% RSLogix 500 project GILL ONION_11_12_2021_BAK142.RSS, saved by version 11.00.00.00 %
PROJECT "UNTITLED"    % processor: MicroLogix 1400 %

PROGRAM FILES
  LAD 2 "MAIN"  10 rungs
  LAD 3 "UNSTACKER"  32 rungs
  LAD 4 "BS"  36 rungs
  LAD 5 "STACKER"  32 rungs
  LAD 6 "WATER"  21 rungs
  LAD 7 "CONVEYORS"  1 rungs
  LAD 8 "ENCODER"  6 rungs  % Bin Scrubber HSC %
  LAD 9 "STARTUP"  6 rungs
  LAD 10 "FAULTS"  65 rungs  % Faults %
  LAD 11 "HSC"  2 rungs  % Bin Scrubber Cradle %

DATA FILES
  O0 OUTPUT  8 elements
  I1 INPUT  18 elements
  S2 STATUS  66 elements
  B3 BINARY  9 elements
  T4 TIMER  34 elements
  C5 COUNTER  1 elements
  R6 CONTROL  1 elements
  N7 INTEGER  21 elements
  F8 FLOAT  1 elements
  L9   3 elements

LADDER 2 "MAIN"
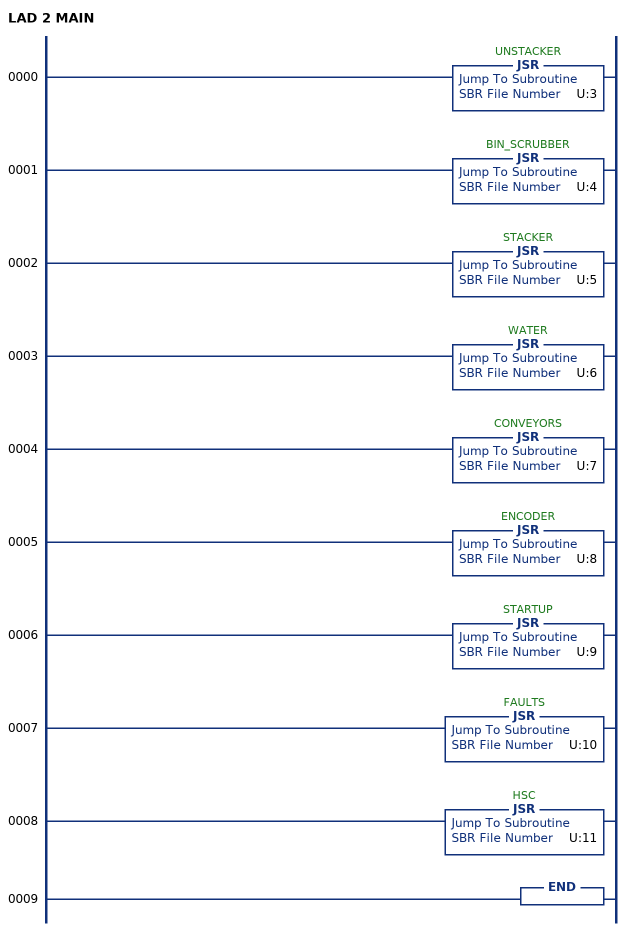
% Rung: 0 %
SOR JSR U:3 EOR
%   U:3  UNSTACKER %
% Rung: 1 %
SOR JSR U:4 EOR
%   U:4  BIN_SCRUBBER %
% Rung: 2 %
SOR JSR U:5 EOR
%   U:5  STACKER %
% Rung: 3 %
SOR JSR U:6 EOR
%   U:6  WATER %
% Rung: 4 %
SOR JSR U:7 EOR
%   U:7  CONVEYORS %
% Rung: 5 %
SOR JSR U:8 EOR
%   U:8  ENCODER %
% Rung: 6 %
SOR JSR U:9 EOR
%   U:9  STARTUP %
% Rung: 7 %
SOR JSR U:10 EOR
%   U:10  FAULTS %
% Rung: 8 %
SOR JSR U:11 EOR
%   U:11  HSC %
% Rung: 9 %
SOR END EOR

LADDER 3 "UNSTACKER"
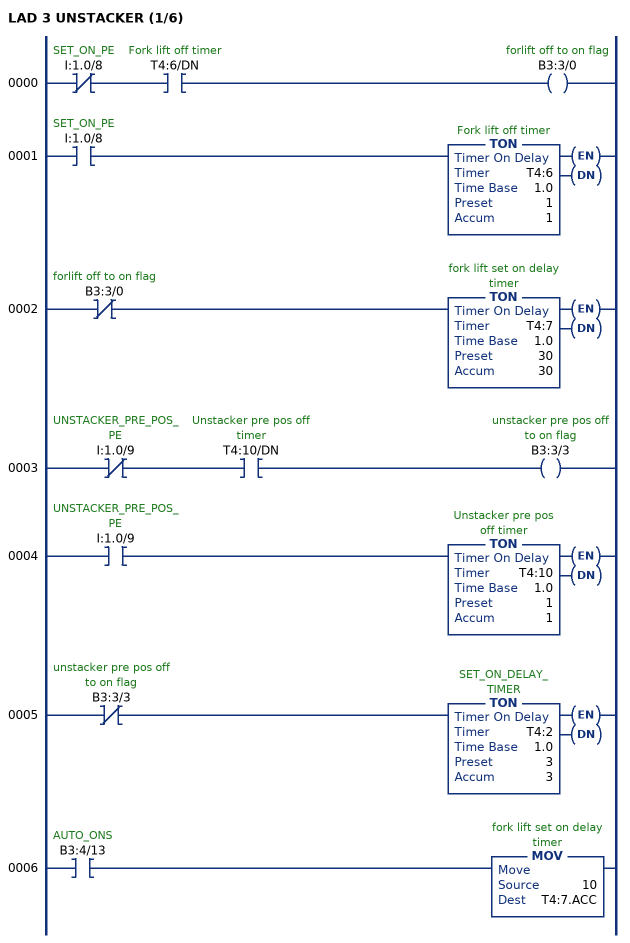
% Rung: 0 %
SOR XIO I:1.0/8 XIC T4:6/DN OTE B3:3/0 EOR
%   I:1.0/8  SET_ON_PE %
%   T4:6  "Fork lift off timer" %
%   B3:3/0  "forlift off to on flag" %
% Rung: 1 %
SOR XIC I:1.0/8 TON T4:6 1.0 1 1 EOR
%   I:1.0/8  SET_ON_PE %
%   T4:6  "Fork lift off timer" %
% Rung: 2 %
SOR XIO B3:3/0 TON T4:7 1.0 30 30 EOR
%   B3:3/0  "forlift off to on flag" %
%   T4:7  "fork lift set on delay timer" %
% Rung: 3 %
SOR XIO I:1.0/9 XIC T4:10/DN OTE B3:3/3 EOR
%   I:1.0/9  UNSTACKER_PRE_POS_PE %
%   T4:10  "Unstacker pre pos off timer" %
%   B3:3/3  "unstacker pre pos off to on flag" %
% Rung: 4 %
SOR XIC I:1.0/9 TON T4:10 1.0 1 1 EOR
%   I:1.0/9  UNSTACKER_PRE_POS_PE %
%   T4:10  "Unstacker pre pos off timer" %
% Rung: 5 %
SOR XIO B3:3/3 TON T4:2 1.0 3 3 EOR
%   B3:3/3  "unstacker pre pos off to on flag" %
%   T4:2  SET_ON_DELAY_TIMER %
% Rung: 6 %
SOR XIC B3:4/13 MOV 10 T4:7.ACC EOR
%   B3:4/13  AUTO_ONS %
%   T4:7  "fork lift set on delay timer" %

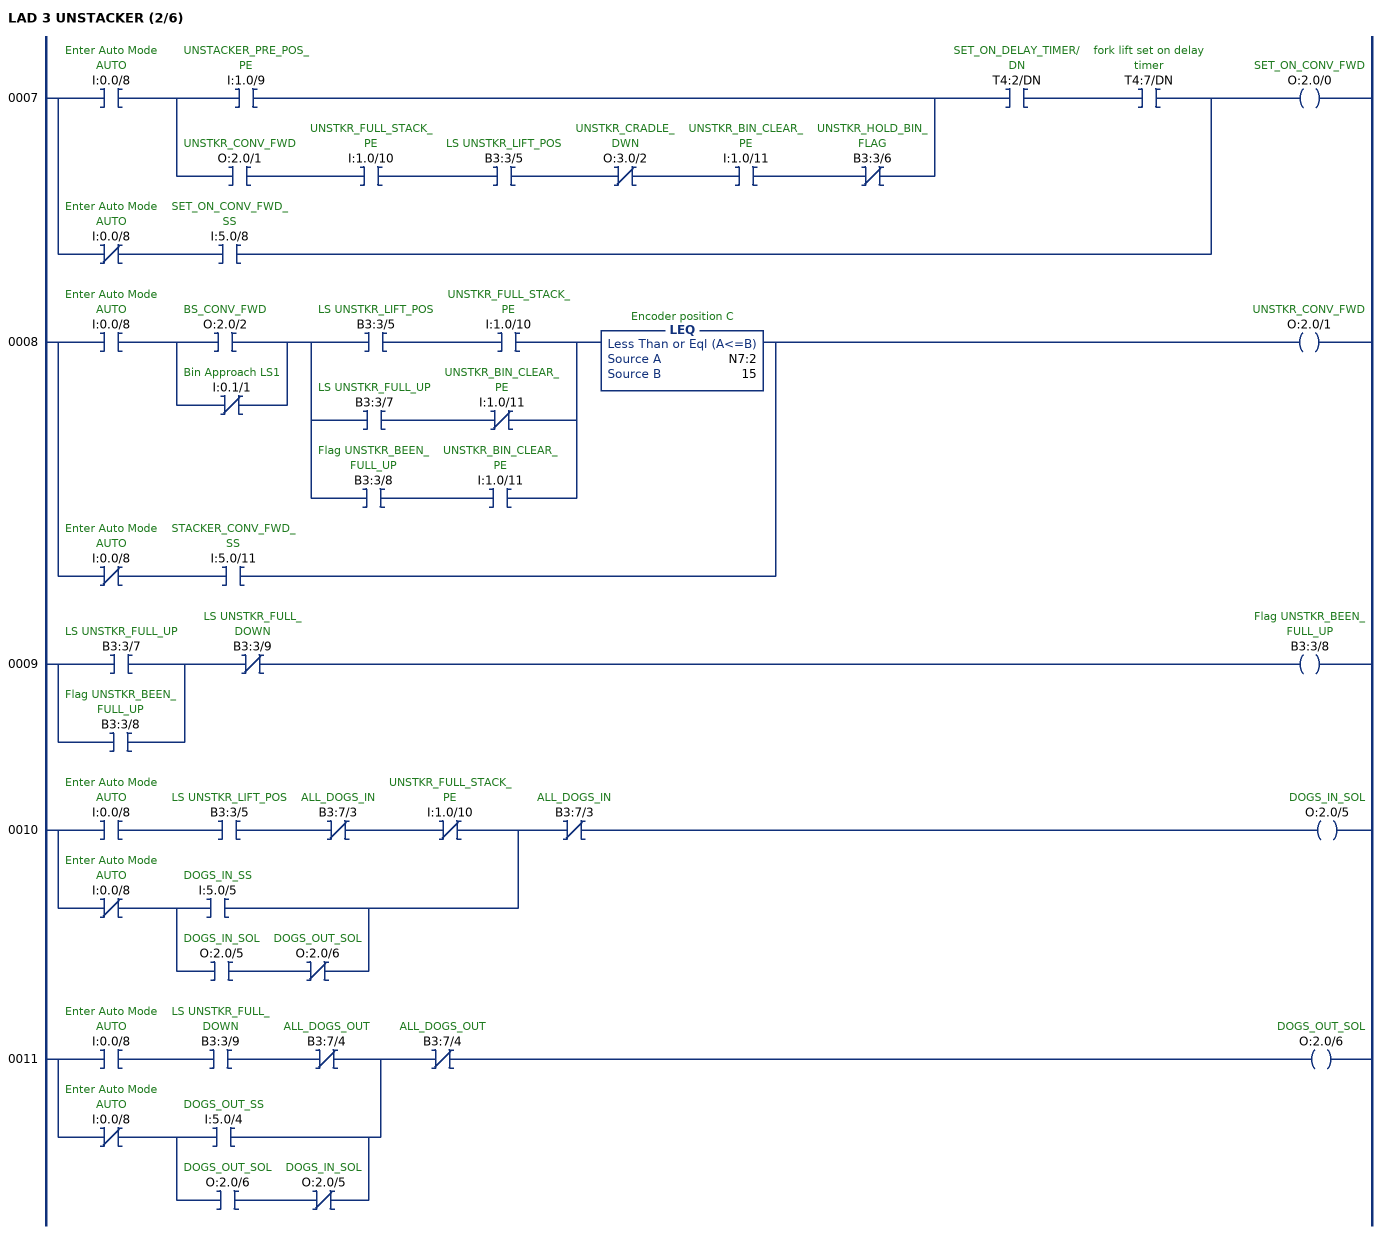
% Rung: 7 %
SOR BST XIC I:0.0/8 BST XIC I:1.0/9 NXB XIC O:2.0/1 XIC I:1.0/10 XIC B3:3/5 XIO O:3.0/2 XIC I:1.0/11 XIO B3:3/6 BND XIC T4:2/DN XIC T4:7/DN NXB XIO I:0.0/8 XIC I:5.0/8 BND OTE O:2.0/0 EOR
%   I:0.0/8  AUTO  "Enter Auto Mode" %
%   I:1.0/9  UNSTACKER_PRE_POS_PE %
%   O:2.0/1  UNSTKR_CONV_FWD %
%   I:1.0/10  UNSTKR_FULL_STACK_PE %
%   B3:3/5  UNSTKR_LIFT_POS  "LS" %
%   O:3.0/2  UNSTKR_CRADLE_DWN %
%   I:1.0/11  UNSTKR_BIN_CLEAR_PE %
%   B3:3/6  UNSTKR_HOLD_BIN_FLAG %
%   T4:2  SET_ON_DELAY_TIMER %
%   T4:7  "fork lift set on delay timer" %
%   I:5.0/8  SET_ON_CONV_FWD_SS %
%   O:2.0/0  SET_ON_CONV_FWD %
% Rung: 8 %
SOR BST XIC I:0.0/8 BST XIC O:2.0/2 NXB XIO I:0.1/1 BND BST XIC B3:3/5 XIC I:1.0/10 NXB BST XIC B3:3/7 XIO I:1.0/11 NXB XIC B3:3/8 XIC I:1.0/11 BND BND LEQ N7:2 15 NXB XIO I:0.0/8 XIC I:5.0/11 BND OTE O:2.0/1 EOR
%   I:0.0/8  AUTO  "Enter Auto Mode" %
%   O:2.0/2  BS_CONV_FWD %
%   I:0.1/1  LS1  "Bin Approach" %
%   B3:3/5  UNSTKR_LIFT_POS  "LS" %
%   I:1.0/10  UNSTKR_FULL_STACK_PE %
%   B3:3/7  UNSTKR_FULL_UP  "LS" %
%   I:1.0/11  UNSTKR_BIN_CLEAR_PE %
%   B3:3/8  UNSTKR_BEEN_FULL_UP  "Flag" %
%   N7:2  C  "Encoder position" %
%   I:5.0/11  STACKER_CONV_FWD_SS %
%   O:2.0/1  UNSTKR_CONV_FWD %
% Rung: 9 %
SOR BST XIC B3:3/7 NXB XIC B3:3/8 BND XIO B3:3/9 OTE B3:3/8 EOR
%   B3:3/7  UNSTKR_FULL_UP  "LS" %
%   B3:3/8  UNSTKR_BEEN_FULL_UP  "Flag" %
%   B3:3/9  UNSTKR_FULL_DOWN  "LS" %
% Rung: 10 %
SOR BST XIC I:0.0/8 XIC B3:3/5 XIO B3:7/3 XIO I:1.0/10 NXB XIO I:0.0/8 BST XIC I:5.0/5 NXB XIC O:2.0/5 XIO O:2.0/6 BND BND XIO B3:7/3 OTE O:2.0/5 EOR
%   I:0.0/8  AUTO  "Enter Auto Mode" %
%   B3:3/5  UNSTKR_LIFT_POS  "LS" %
%   B3:7/3  ALL_DOGS_IN %
%   I:1.0/10  UNSTKR_FULL_STACK_PE %
%   I:5.0/5  DOGS_IN_SS %
%   O:2.0/5  DOGS_IN_SOL %
%   O:2.0/6  DOGS_OUT_SOL %
% Rung: 11 %
SOR BST XIC I:0.0/8 XIC B3:3/9 XIO B3:7/4 NXB XIO I:0.0/8 BST XIC I:5.0/4 NXB XIC O:2.0/6 XIO O:2.0/5 BND BND XIO B3:7/4 OTE O:2.0/6 EOR
%   I:0.0/8  AUTO  "Enter Auto Mode" %
%   B3:3/9  UNSTKR_FULL_DOWN  "LS" %
%   B3:7/4  ALL_DOGS_OUT %
%   I:5.0/4  DOGS_OUT_SS %
%   O:2.0/6  DOGS_OUT_SOL %
%   O:2.0/5  DOGS_IN_SOL %

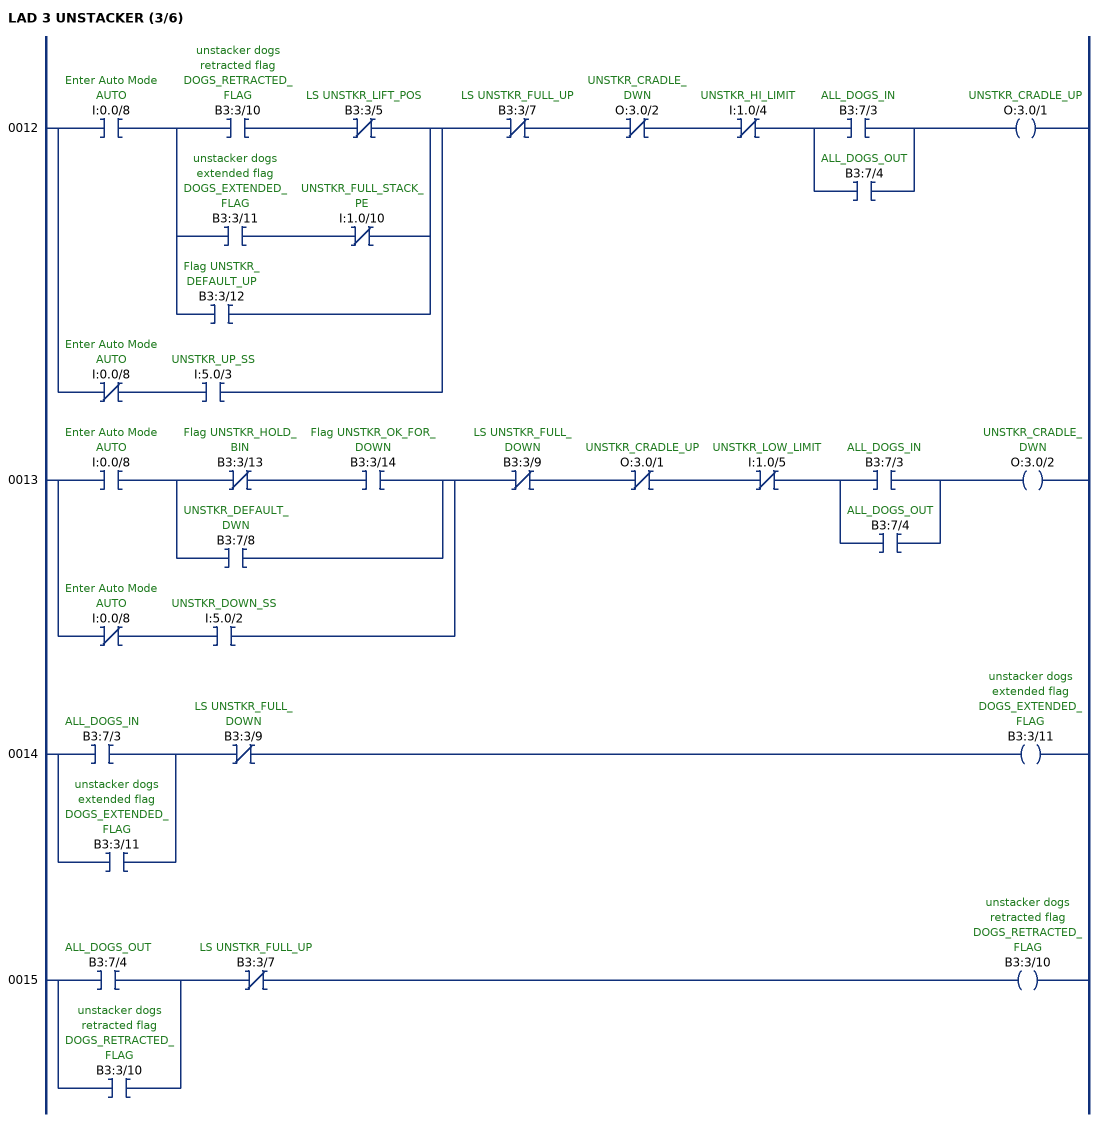
% Rung: 12 %
SOR BST XIC I:0.0/8 BST XIC B3:3/10 XIO B3:3/5 NXB BST XIC B3:3/11 XIO I:1.0/10 NXB XIC B3:3/12 BND BND NXB XIO I:0.0/8 XIC I:5.0/3 BND XIO B3:3/7 XIO O:3.0/2 XIO I:1.0/4 BST XIC B3:7/3 NXB XIC B3:7/4 BND OTE O:3.0/1 EOR
%   I:0.0/8  AUTO  "Enter Auto Mode" %
%   B3:3/10  DOGS_RETRACTED_FLAG  "unstacker dogs retracted flag" %
%   B3:3/5  UNSTKR_LIFT_POS  "LS" %
%   B3:3/11  DOGS_EXTENDED_FLAG  "unstacker dogs extended flag" %
%   I:1.0/10  UNSTKR_FULL_STACK_PE %
%   B3:3/12  UNSTKR_DEFAULT_UP  "Flag" %
%   I:5.0/3  UNSTKR_UP_SS %
%   B3:3/7  UNSTKR_FULL_UP  "LS" %
%   O:3.0/2  UNSTKR_CRADLE_DWN %
%   I:1.0/4  UNSTKR_HI_LIMIT %
%   B3:7/3  ALL_DOGS_IN %
%   B3:7/4  ALL_DOGS_OUT %
%   O:3.0/1  UNSTKR_CRADLE_UP %
% Rung: 13 %
SOR BST XIC I:0.0/8 BST XIO B3:3/13 XIC B3:3/14 NXB XIC B3:7/8 BND NXB XIO I:0.0/8 XIC I:5.0/2 BND XIO B3:3/9 XIO O:3.0/1 XIO I:1.0/5 BST XIC B3:7/3 NXB XIC B3:7/4 BND OTE O:3.0/2 EOR
%   I:0.0/8  AUTO  "Enter Auto Mode" %
%   B3:3/13  UNSTKR_HOLD_BIN  "Flag" %
%   B3:3/14  UNSTKR_OK_FOR_DOWN  "Flag" %
%   B3:7/8  UNSTKR_DEFAULT_DWN %
%   I:5.0/2  UNSTKR_DOWN_SS %
%   B3:3/9  UNSTKR_FULL_DOWN  "LS" %
%   O:3.0/1  UNSTKR_CRADLE_UP %
%   I:1.0/5  UNSTKR_LOW_LIMIT %
%   B3:7/3  ALL_DOGS_IN %
%   B3:7/4  ALL_DOGS_OUT %
%   O:3.0/2  UNSTKR_CRADLE_DWN %
% Rung: 14 %
SOR BST XIC B3:7/3 NXB XIC B3:3/11 BND XIO B3:3/9 OTE B3:3/11 EOR
%   B3:7/3  ALL_DOGS_IN %
%   B3:3/11  DOGS_EXTENDED_FLAG  "unstacker dogs extended flag" %
%   B3:3/9  UNSTKR_FULL_DOWN  "LS" %
% Rung: 15 %
SOR BST XIC B3:7/4 NXB XIC B3:3/10 BND XIO B3:3/7 OTE B3:3/10 EOR
%   B3:7/4  ALL_DOGS_OUT %
%   B3:3/10  DOGS_RETRACTED_FLAG  "unstacker dogs retracted flag" %
%   B3:3/7  UNSTKR_FULL_UP  "LS" %

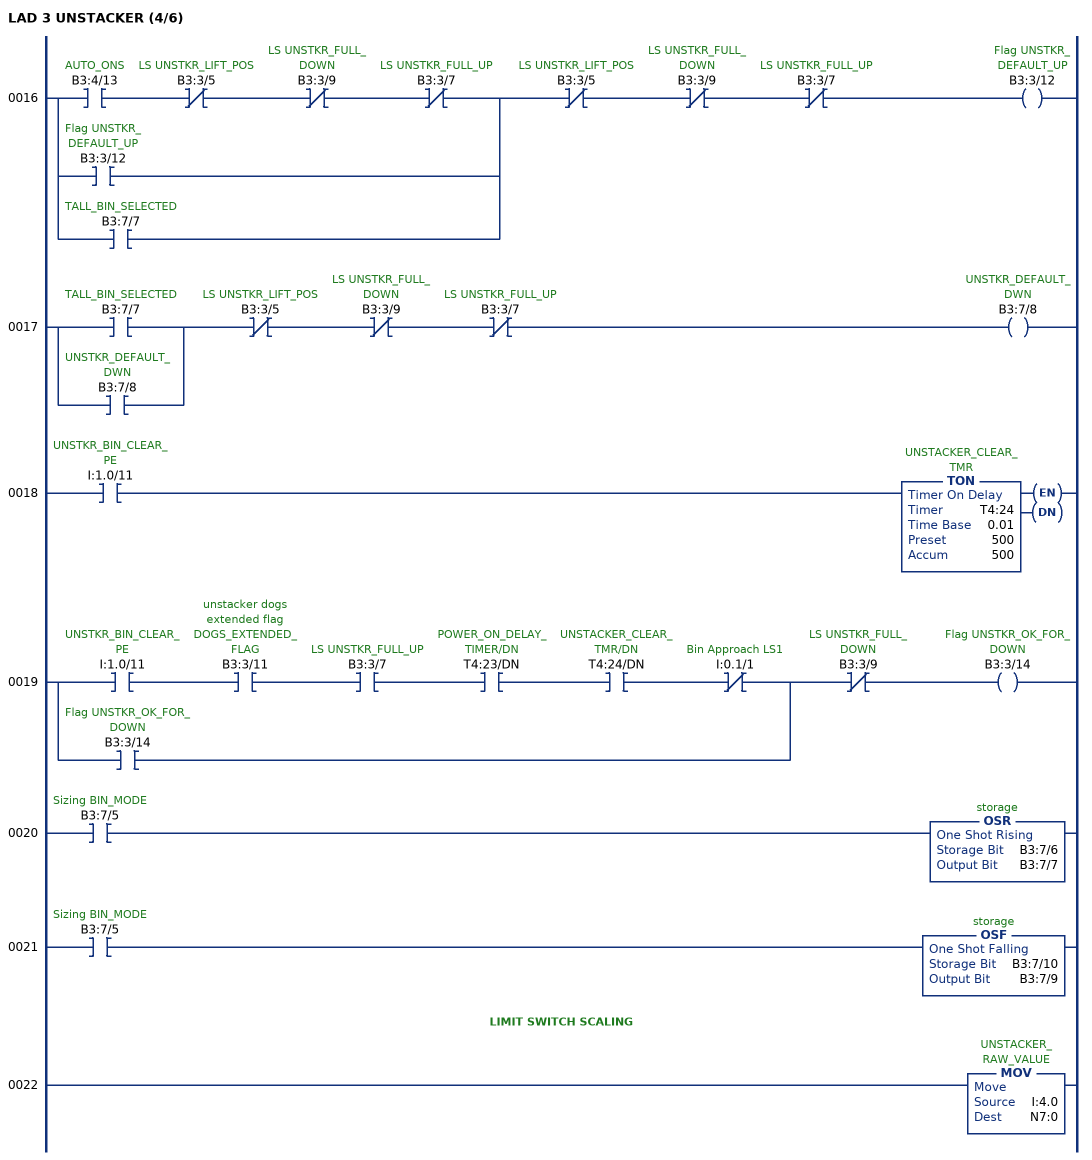
% Rung: 16 %
SOR BST XIC B3:4/13 XIO B3:3/5 XIO B3:3/9 XIO B3:3/7 NXB BST XIC B3:3/12 NXB XIC B3:7/7 BND BND XIO B3:3/5 XIO B3:3/9 XIO B3:3/7 OTE B3:3/12 EOR
%   B3:4/13  AUTO_ONS %
%   B3:3/5  UNSTKR_LIFT_POS  "LS" %
%   B3:3/9  UNSTKR_FULL_DOWN  "LS" %
%   B3:3/7  UNSTKR_FULL_UP  "LS" %
%   B3:3/12  UNSTKR_DEFAULT_UP  "Flag" %
%   B3:7/7  TALL_BIN_SELECTED %
% Rung: 17 %
SOR BST XIC B3:7/7 NXB XIC B3:7/8 BND XIO B3:3/5 XIO B3:3/9 XIO B3:3/7 OTE B3:7/8 EOR
%   B3:7/7  TALL_BIN_SELECTED %
%   B3:7/8  UNSTKR_DEFAULT_DWN %
%   B3:3/5  UNSTKR_LIFT_POS  "LS" %
%   B3:3/9  UNSTKR_FULL_DOWN  "LS" %
%   B3:3/7  UNSTKR_FULL_UP  "LS" %
% Rung: 18 %
SOR XIC I:1.0/11 TON T4:24 0.01 500 500 EOR
%   I:1.0/11  UNSTKR_BIN_CLEAR_PE %
%   T4:24  UNSTACKER_CLEAR_TMR %
% Rung: 19 %
SOR BST XIC I:1.0/11 XIC B3:3/11 XIC B3:3/7 XIC T4:23/DN XIC T4:24/DN XIO I:0.1/1 NXB XIC B3:3/14 BND XIO B3:3/9 OTE B3:3/14 EOR
%   I:1.0/11  UNSTKR_BIN_CLEAR_PE %
%   B3:3/11  DOGS_EXTENDED_FLAG  "unstacker dogs extended flag" %
%   B3:3/7  UNSTKR_FULL_UP  "LS" %
%   T4:23  POWER_ON_DELAY_TIMER %
%   T4:24  UNSTACKER_CLEAR_TMR %
%   I:0.1/1  LS1  "Bin Approach" %
%   B3:3/14  UNSTKR_OK_FOR_DOWN  "Flag" %
%   B3:3/9  UNSTKR_FULL_DOWN  "LS" %
% Rung: 20 %
SOR XIC B3:7/5 OSR B3:7/6 B3:7/7 EOR
%   B3:7/5  BIN_MODE  "Sizing" %
%   B3:7/6  "storage" %
%   B3:7/7  TALL_BIN_SELECTED %
% Rung: 21 %
SOR XIC B3:7/5 OSF B3:7/10 B3:7/9 EOR
%   B3:7/5  BIN_MODE  "Sizing" %
%   B3:7/10  "storage" %
%   B3:7/9  SMALL_BIN_SELECTED %
% Rung: 22 %
% TITLE: LIMIT SWITCH SCALING %
SOR MOV I:4.0 N7:0 EOR
%   I:4.0  UNSTACKER_RAW  "Draw String Encoder" %
%   N7:0  UNSTACKER_RAW_VALUE %

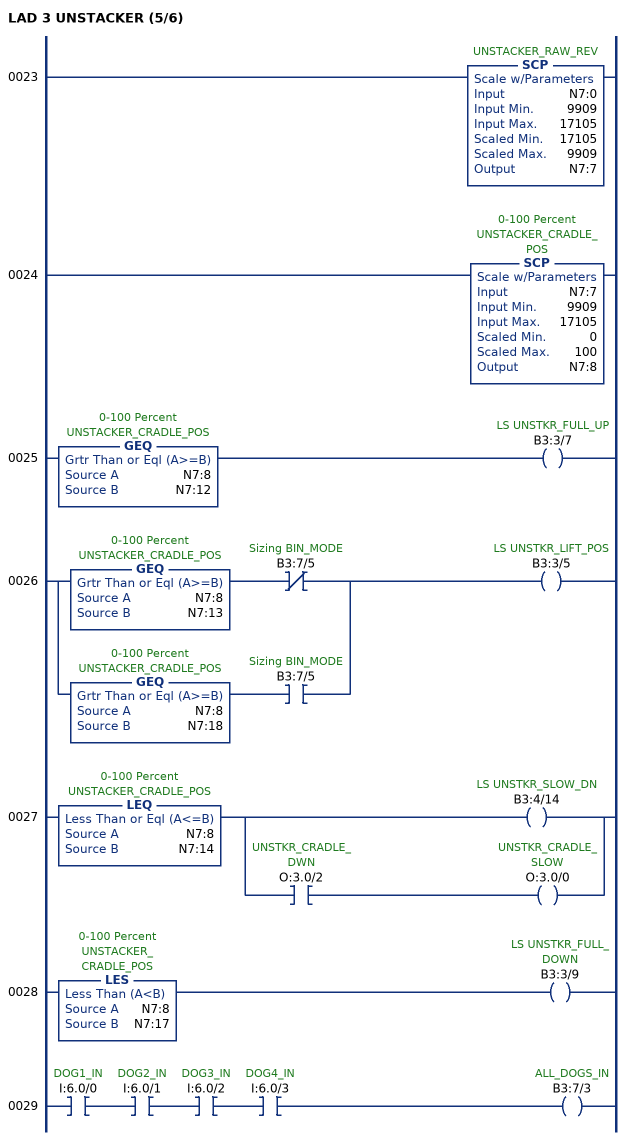
% Rung: 23 %
SOR SCP N7:0 9909 17105 17105 9909 N7:7 EOR
%   N7:0  UNSTACKER_RAW_VALUE %
%   N7:7  UNSTACKER_RAW_REV %
% Rung: 24 %
SOR SCP N7:7 9909 17105 0 100 N7:8 EOR
%   N7:7  UNSTACKER_RAW_REV %
%   N7:8  UNSTACKER_CRADLE_POS  "0-100 Percent" %
% Rung: 25 %
SOR GEQ N7:8 N7:12 OTE B3:3/7 EOR
%   N7:8  UNSTACKER_CRADLE_POS  "0-100 Percent" %
%   N7:12  UNSTKR_FULL_UP_SP  "Unstacker" %
%   B3:3/7  UNSTKR_FULL_UP  "LS" %
% Rung: 26 %
SOR BST GEQ N7:8 N7:13 XIO B3:7/5 NXB GEQ N7:8 N7:18 XIC B3:7/5 BND OTE B3:3/5 EOR
%   N7:8  UNSTACKER_CRADLE_POS  "0-100 Percent" %
%   N7:13  UNSTACKER_LIFT_SP  "Unstacker Lift Pos" %
%   B3:7/5  BIN_MODE  "Sizing" %
%   N7:18  TALL_BIN_SP %
%   B3:3/5  UNSTKR_LIFT_POS  "LS" %
% Rung: 27 %
SOR LEQ N7:8 N7:14 BST OTE B3:4/14 NXB XIC O:3.0/2 OTE O:3.0/0 BND EOR
%   N7:8  UNSTACKER_CRADLE_POS  "0-100 Percent" %
%   N7:14  UNSTKR_FULL_DOWN_SP  "Unstacker Full Down" %
%   B3:4/14  UNSTKR_SLOW_DN  "LS" %
%   O:3.0/2  UNSTKR_CRADLE_DWN %
%   O:3.0/0  UNSTKR_CRADLE_SLOW %
% Rung: 28 %
SOR LES N7:8 N7:17 OTE B3:3/9 EOR
%   N7:8  UNSTACKER_CRADLE_POS  "0-100 Percent" %
%   N7:17  "Unstacker" %
%   B3:3/9  UNSTKR_FULL_DOWN  "LS" %
% Rung: 29 %
SOR XIC I:6.0/0 XIC I:6.0/1 XIC I:6.0/2 XIC I:6.0/3 OTE B3:7/3 EOR
%   I:6.0/0  DOG1_IN %
%   I:6.0/1  DOG2_IN %
%   I:6.0/2  DOG3_IN %
%   I:6.0/3  DOG4_IN %
%   B3:7/3  ALL_DOGS_IN %

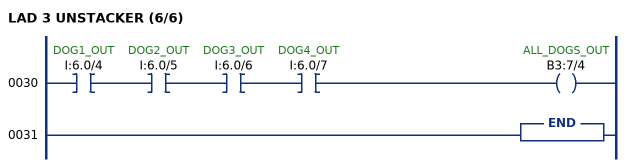
% Rung: 30 %
SOR XIC I:6.0/4 XIC I:6.0/5 XIC I:6.0/6 XIC I:6.0/7 OTE B3:7/4 EOR
%   I:6.0/4  DOG1_OUT %
%   I:6.0/5  DOG2_OUT %
%   I:6.0/6  DOG3_OUT %
%   I:6.0/7  DOG4_OUT %
%   B3:7/4  ALL_DOGS_OUT %
% Rung: 31 %
SOR END EOR

LADDER 4 "BS"
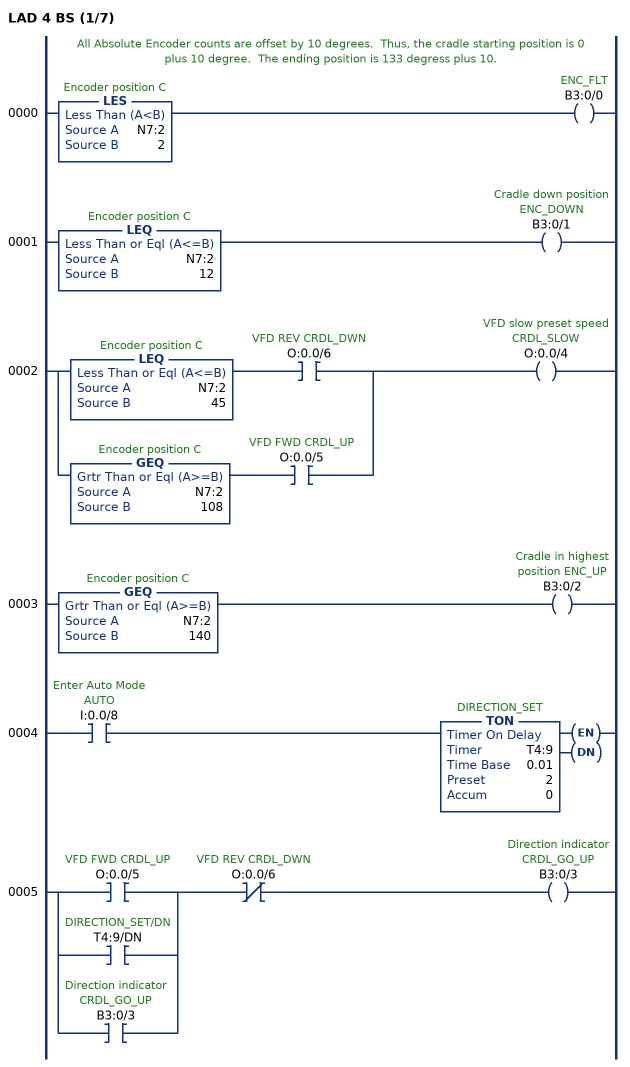
% Rung: 0 %
% All Absolute Encoder counts are offset by 10 degrees.  Thus, the cradle starting position is 0 plus 10 degree.  The ending position is 133 degress plus 10. %
SOR LES N7:2 2 OTE B3:0/0 EOR
%   N7:2  C  "Encoder position" %
%   B3:0/0  ENC_FLT %
% Rung: 1 %
SOR LEQ N7:2 12 OTE B3:0/1 EOR
%   N7:2  C  "Encoder position" %
%   B3:0/1  ENC_DOWN  "Cradle down position" %
% Rung: 2 %
SOR BST LEQ N7:2 45 XIC O:0.0/6 NXB GEQ N7:2 108 XIC O:0.0/5 BND OTE O:0.0/4 EOR
%   N7:2  C  "Encoder position" %
%   O:0.0/6  CRDL_DWN  "VFD REV" %
%   O:0.0/5  CRDL_UP  "VFD FWD" %
%   O:0.0/4  CRDL_SLOW  "VFD slow preset speed" %
% Rung: 3 %
SOR GEQ N7:2 140 OTE B3:0/2 EOR
%   N7:2  C  "Encoder position" %
%   B3:0/2  ENC_UP  "Cradle in highest position" %
% Rung: 4 %
SOR XIC I:0.0/8 TON T4:9 0.01 2 0 EOR
%   I:0.0/8  AUTO  "Enter Auto Mode" %
%   T4:9  DIRECTION_SET %
% Rung: 5 %
SOR BST XIC O:0.0/5 NXB XIC T4:9/DN NXB XIC B3:0/3 BND XIO O:0.0/6 OTE B3:0/3 EOR
%   O:0.0/5  CRDL_UP  "VFD FWD" %
%   T4:9  DIRECTION_SET %
%   B3:0/3  CRDL_GO_UP  "Direction indicator" %
%   O:0.0/6  CRDL_DWN  "VFD REV" %

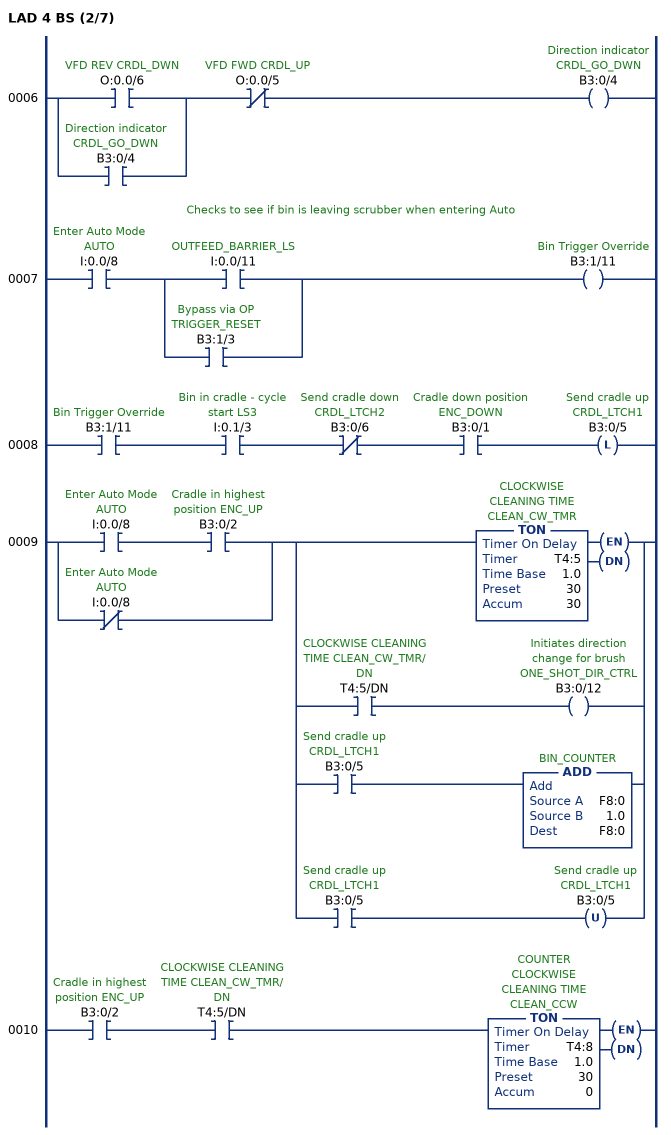
% Rung: 6 %
SOR BST XIC O:0.0/6 NXB XIC B3:0/4 BND XIO O:0.0/5 OTE B3:0/4 EOR
%   O:0.0/6  CRDL_DWN  "VFD REV" %
%   B3:0/4  CRDL_GO_DWN  "Direction indicator" %
%   O:0.0/5  CRDL_UP  "VFD FWD" %
% Rung: 7 %
% Checks to see if bin is leaving scrubber when entering Auto %
SOR XIC I:0.0/8 BST XIC I:0.0/11 NXB XIC B3:1/3 BND OTE B3:1/11 EOR
%   I:0.0/8  AUTO  "Enter Auto Mode" %
%   I:0.0/11  OUTFEED_BARRIER_LS %
%   B3:1/3  TRIGGER_RESET  "Bypass via OP" %
%   B3:1/11  "Bin Trigger Override" %
% Rung: 8 %
SOR XIC B3:1/11 XIC I:0.1/3 XIO B3:0/6 XIC B3:0/1 OTL B3:0/5 EOR
%   B3:1/11  "Bin Trigger Override" %
%   I:0.1/3  LS3  "Bin in cradle - cycle start" %
%   B3:0/6  CRDL_LTCH2  "Send cradle down" %
%   B3:0/1  ENC_DOWN  "Cradle down position" %
%   B3:0/5  CRDL_LTCH1  "Send cradle up" %
% Rung: 9 %
SOR BST XIC I:0.0/8 XIC B3:0/2 NXB XIO I:0.0/8 BND BST TON T4:5 1.0 30 30 NXB XIC T4:5/DN OTE B3:0/12 NXB BST XIC B3:0/5 ADD F8:0 1.0 F8:0 NXB XIC B3:0/5 OTU B3:0/5 BND BND EOR
%   I:0.0/8  AUTO  "Enter Auto Mode" %
%   B3:0/2  ENC_UP  "Cradle in highest position" %
%   T4:5  CLEAN_CW_TMR  "CLOCKWISE CLEANING TIME" %
%   B3:0/12  ONE_SHOT_DIR_CTRL  "Initiates direction change for brush" %
%   B3:0/5  CRDL_LTCH1  "Send cradle up" %
%   F8:0  BIN_COUNTER %
% Rung: 10 %
SOR XIC B3:0/2 XIC T4:5/DN TON T4:8 1.0 30 0 EOR
%   B3:0/2  ENC_UP  "Cradle in highest position" %
%   T4:5  CLEAN_CW_TMR  "CLOCKWISE CLEANING TIME" %
%   T4:8  CLEAN_CCW  "COUNTER CLOCKWISE CLEANING TIME" %

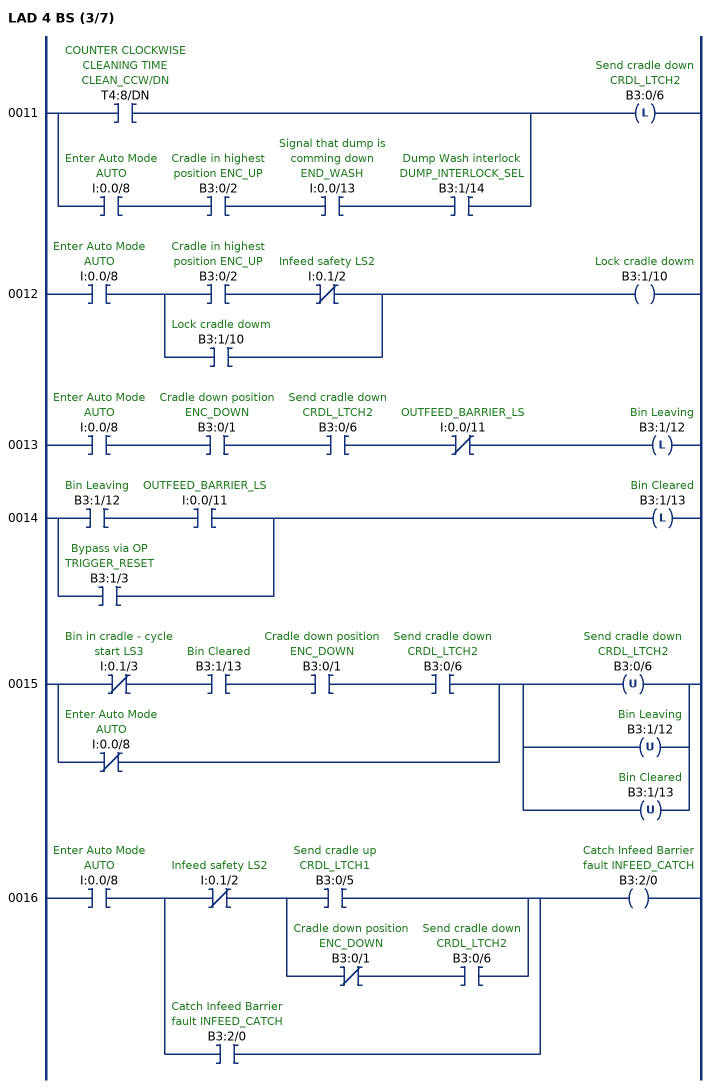
% Rung: 11 %
SOR BST XIC T4:8/DN NXB XIC I:0.0/8 XIC B3:0/2 XIC I:0.0/13 XIC B3:1/14 BND OTL B3:0/6 EOR
%   T4:8  CLEAN_CCW  "COUNTER CLOCKWISE CLEANING TIME" %
%   I:0.0/8  AUTO  "Enter Auto Mode" %
%   B3:0/2  ENC_UP  "Cradle in highest position" %
%   I:0.0/13  END_WASH  "Signal that dump is comming down" %
%   B3:1/14  DUMP_INTERLOCK_SEL  "Dump Wash interlock" %
%   B3:0/6  CRDL_LTCH2  "Send cradle down" %
% Rung: 12 %
SOR XIC I:0.0/8 BST XIC B3:0/2 XIO I:0.1/2 NXB XIC B3:1/10 BND OTE B3:1/10 EOR
%   I:0.0/8  AUTO  "Enter Auto Mode" %
%   B3:0/2  ENC_UP  "Cradle in highest position" %
%   I:0.1/2  LS2  "Infeed safety" %
%   B3:1/10  "Lock cradle dowm" %
% Rung: 13 %
SOR XIC I:0.0/8 XIC B3:0/1 XIC B3:0/6 XIO I:0.0/11 OTL B3:1/12 EOR
%   I:0.0/8  AUTO  "Enter Auto Mode" %
%   B3:0/1  ENC_DOWN  "Cradle down position" %
%   B3:0/6  CRDL_LTCH2  "Send cradle down" %
%   I:0.0/11  OUTFEED_BARRIER_LS %
%   B3:1/12  "Bin Leaving" %
% Rung: 14 %
SOR BST XIC B3:1/12 XIC I:0.0/11 NXB XIC B3:1/3 BND OTL B3:1/13 EOR
%   B3:1/12  "Bin Leaving" %
%   I:0.0/11  OUTFEED_BARRIER_LS %
%   B3:1/3  TRIGGER_RESET  "Bypass via OP" %
%   B3:1/13  "Bin Cleared" %
% Rung: 15 %
SOR BST XIO I:0.1/3 XIC B3:1/13 XIC B3:0/1 XIC B3:0/6 NXB XIO I:0.0/8 BND BST OTU B3:0/6 NXB BST OTU B3:1/12 NXB OTU B3:1/13 BND BND EOR
%   I:0.1/3  LS3  "Bin in cradle - cycle start" %
%   B3:1/13  "Bin Cleared" %
%   B3:0/1  ENC_DOWN  "Cradle down position" %
%   B3:0/6  CRDL_LTCH2  "Send cradle down" %
%   I:0.0/8  AUTO  "Enter Auto Mode" %
%   B3:1/12  "Bin Leaving" %
% Rung: 16 %
SOR XIC I:0.0/8 BST XIO I:0.1/2 BST XIC B3:0/5 NXB XIO B3:0/1 XIC B3:0/6 BND NXB XIC B3:2/0 BND OTE B3:2/0 EOR
%   I:0.0/8  AUTO  "Enter Auto Mode" %
%   I:0.1/2  LS2  "Infeed safety" %
%   B3:0/5  CRDL_LTCH1  "Send cradle up" %
%   B3:0/1  ENC_DOWN  "Cradle down position" %
%   B3:0/6  CRDL_LTCH2  "Send cradle down" %
%   B3:2/0  INFEED_CATCH  "Catch Infeed Barrier fault" %

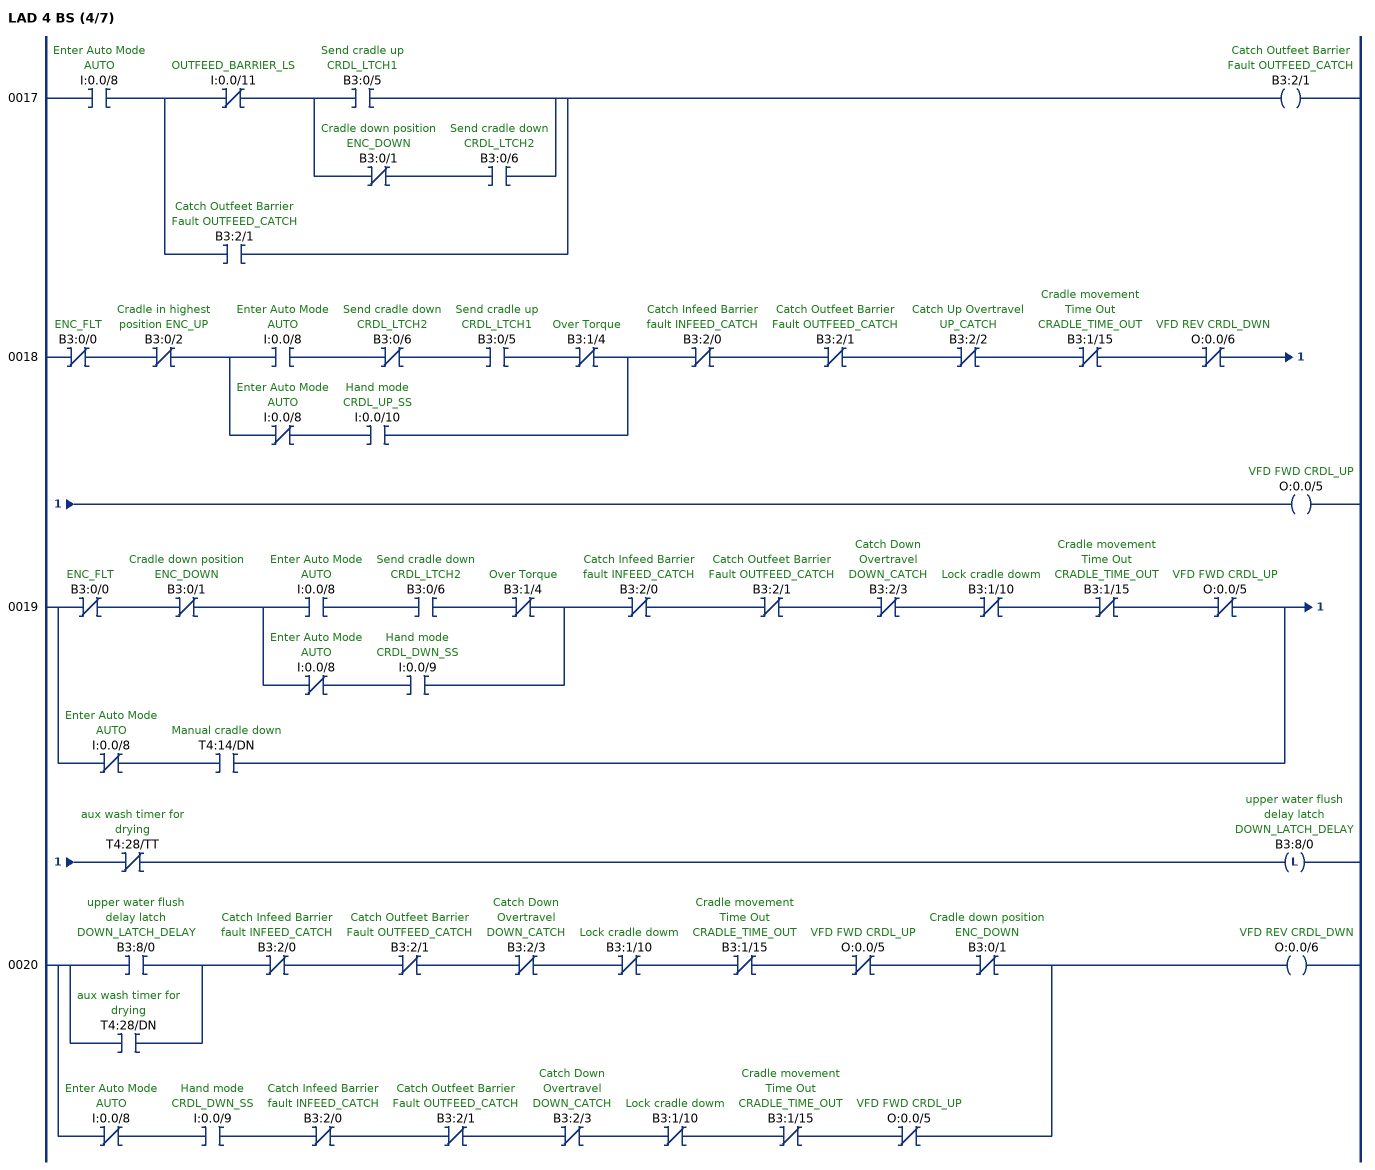
% Rung: 17 %
SOR XIC I:0.0/8 BST XIO I:0.0/11 BST XIC B3:0/5 NXB XIO B3:0/1 XIC B3:0/6 BND NXB XIC B3:2/1 BND OTE B3:2/1 EOR
%   I:0.0/8  AUTO  "Enter Auto Mode" %
%   I:0.0/11  OUTFEED_BARRIER_LS %
%   B3:0/5  CRDL_LTCH1  "Send cradle up" %
%   B3:0/1  ENC_DOWN  "Cradle down position" %
%   B3:0/6  CRDL_LTCH2  "Send cradle down" %
%   B3:2/1  OUTFEED_CATCH  "Catch Outfeet Barrier Fault" %
% Rung: 18 %
SOR XIO B3:0/0 XIO B3:0/2 BST XIC I:0.0/8 XIO B3:0/6 XIC B3:0/5 XIO B3:1/4 NXB XIO I:0.0/8 XIC I:0.0/10 BND XIO B3:2/0 XIO B3:2/1 XIO B3:2/2 XIO B3:1/15 XIO O:0.0/6 OTE O:0.0/5 EOR
%   B3:0/0  ENC_FLT %
%   B3:0/2  ENC_UP  "Cradle in highest position" %
%   I:0.0/8  AUTO  "Enter Auto Mode" %
%   B3:0/6  CRDL_LTCH2  "Send cradle down" %
%   B3:0/5  CRDL_LTCH1  "Send cradle up" %
%   B3:1/4  "Over Torque" %
%   I:0.0/10  CRDL_UP_SS  "Hand mode" %
%   B3:2/0  INFEED_CATCH  "Catch Infeed Barrier fault" %
%   B3:2/1  OUTFEED_CATCH  "Catch Outfeet Barrier Fault" %
%   B3:2/2  UP_CATCH  "Catch Up Overtravel" %
%   B3:1/15  CRADLE_TIME_OUT  "Cradle movement Time Out" %
%   O:0.0/6  CRDL_DWN  "VFD REV" %
%   O:0.0/5  CRDL_UP  "VFD FWD" %
% Rung: 19 %
SOR BST XIO B3:0/0 XIO B3:0/1 BST XIC I:0.0/8 XIC B3:0/6 XIO B3:1/4 NXB XIO I:0.0/8 XIC I:0.0/9 BND XIO B3:2/0 XIO B3:2/1 XIO B3:2/3 XIO B3:1/10 XIO B3:1/15 XIO O:0.0/5 NXB XIO I:0.0/8 XIC T4:14/DN BND XIO T4:28/TT OTL B3:8/0 EOR
%   B3:0/0  ENC_FLT %
%   B3:0/1  ENC_DOWN  "Cradle down position" %
%   I:0.0/8  AUTO  "Enter Auto Mode" %
%   B3:0/6  CRDL_LTCH2  "Send cradle down" %
%   B3:1/4  "Over Torque" %
%   I:0.0/9  CRDL_DWN_SS  "Hand mode" %
%   B3:2/0  INFEED_CATCH  "Catch Infeed Barrier fault" %
%   B3:2/1  OUTFEED_CATCH  "Catch Outfeet Barrier Fault" %
%   B3:2/3  DOWN_CATCH  "Catch Down Overtravel" %
%   B3:1/10  "Lock cradle dowm" %
%   B3:1/15  CRADLE_TIME_OUT  "Cradle movement Time Out" %
%   O:0.0/5  CRDL_UP  "VFD FWD" %
%   T4:14  "Manual cradle down" %
%   T4:28  "aux wash timer for drying" %
%   B3:8/0  DOWN_LATCH_DELAY  "upper water flush delay latch" %
% Rung: 20 %
SOR BST BST XIC B3:8/0 NXB XIC T4:28/DN BND XIO B3:2/0 XIO B3:2/1 XIO B3:2/3 XIO B3:1/10 XIO B3:1/15 XIO O:0.0/5 XIO B3:0/1 NXB XIO I:0.0/8 XIC I:0.0/9 XIO B3:2/0 XIO B3:2/1 XIO B3:2/3 XIO B3:1/10 XIO B3:1/15 XIO O:0.0/5 BND OTE O:0.0/6 EOR
%   B3:8/0  DOWN_LATCH_DELAY  "upper water flush delay latch" %
%   T4:28  "aux wash timer for drying" %
%   B3:2/0  INFEED_CATCH  "Catch Infeed Barrier fault" %
%   B3:2/1  OUTFEED_CATCH  "Catch Outfeet Barrier Fault" %
%   B3:2/3  DOWN_CATCH  "Catch Down Overtravel" %
%   B3:1/10  "Lock cradle dowm" %
%   B3:1/15  CRADLE_TIME_OUT  "Cradle movement Time Out" %
%   O:0.0/5  CRDL_UP  "VFD FWD" %
%   B3:0/1  ENC_DOWN  "Cradle down position" %
%   I:0.0/8  AUTO  "Enter Auto Mode" %
%   I:0.0/9  CRDL_DWN_SS  "Hand mode" %
%   O:0.0/6  CRDL_DWN  "VFD REV" %

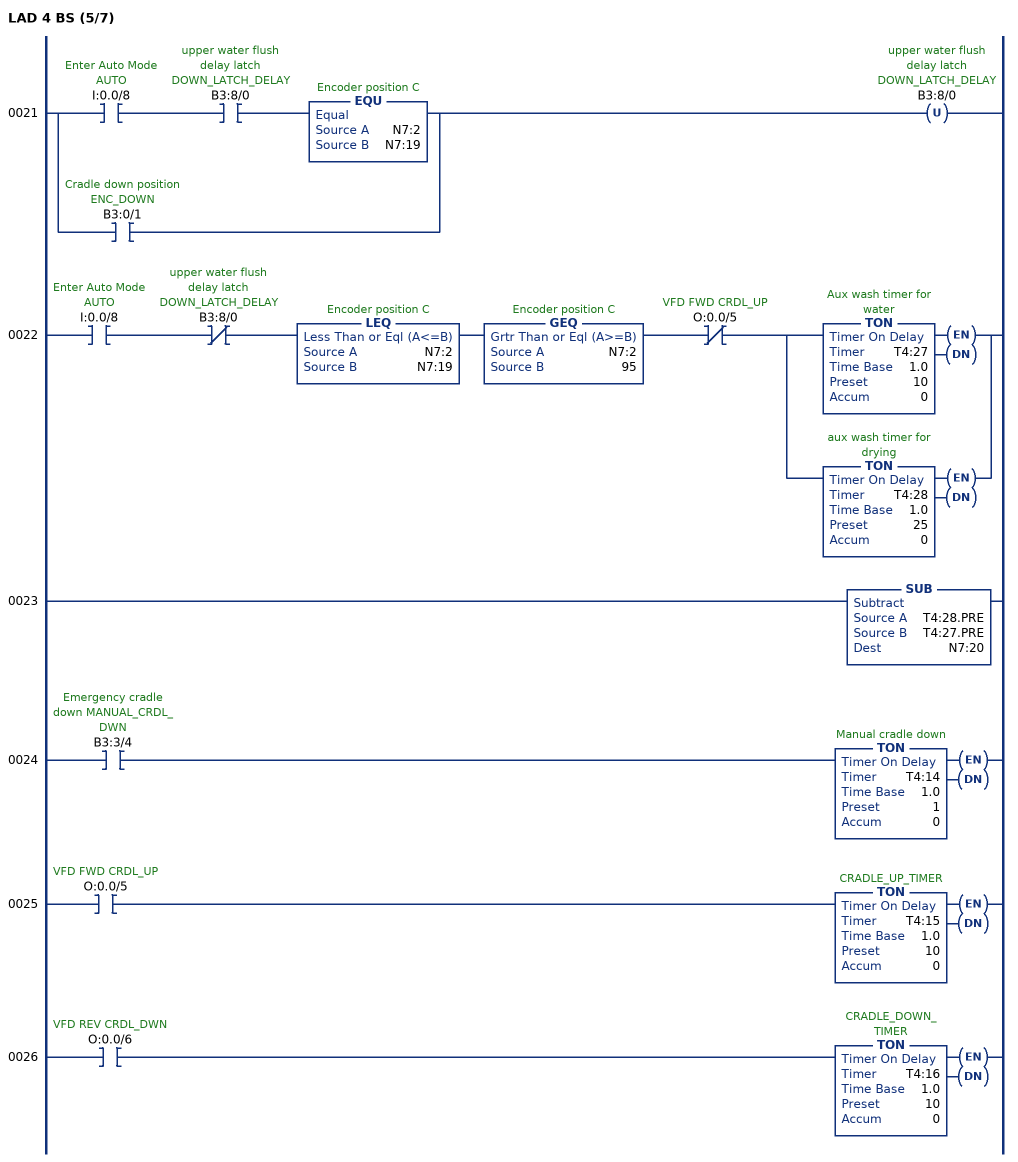
% Rung: 21 %
SOR BST XIC I:0.0/8 XIC B3:8/0 EQU N7:2 N7:19 NXB XIC B3:0/1 BND OTU B3:8/0 EOR
%   I:0.0/8  AUTO  "Enter Auto Mode" %
%   B3:8/0  DOWN_LATCH_DELAY  "upper water flush delay latch" %
%   N7:2  C  "Encoder position" %
%   N7:19  UPPER_WASH_SET_POINT  "HMI input for aux upper wash" %
%   B3:0/1  ENC_DOWN  "Cradle down position" %
% Rung: 22 %
SOR XIC I:0.0/8 XIO B3:8/0 LEQ N7:2 N7:19 GEQ N7:2 95 XIO O:0.0/5 BST TON T4:27 1.0 10 0 NXB TON T4:28 1.0 25 0 BND EOR
%   I:0.0/8  AUTO  "Enter Auto Mode" %
%   B3:8/0  DOWN_LATCH_DELAY  "upper water flush delay latch" %
%   N7:2  C  "Encoder position" %
%   N7:19  UPPER_WASH_SET_POINT  "HMI input for aux upper wash" %
%   O:0.0/5  CRDL_UP  "VFD FWD" %
%   T4:27  "Aux wash timer for water" %
%   T4:28  "aux wash timer for drying" %
% Rung: 23 %
SOR SUB T4:28.PRE T4:27.PRE N7:20 EOR
%   T4:28  "aux wash timer for drying" %
%   T4:27  "Aux wash timer for water" %
% Rung: 24 %
SOR XIC B3:3/4 TON T4:14 1.0 1 0 EOR
%   B3:3/4  MANUAL_CRDL_DWN  "Emergency cradle down" %
%   T4:14  "Manual cradle down" %
% Rung: 25 %
SOR XIC O:0.0/5 TON T4:15 1.0 10 0 EOR
%   O:0.0/5  CRDL_UP  "VFD FWD" %
%   T4:15  CRADLE_UP_TIMER %
% Rung: 26 %
SOR XIC O:0.0/6 TON T4:16 1.0 10 0 EOR
%   O:0.0/6  CRDL_DWN  "VFD REV" %
%   T4:16  CRADLE_DOWN_TIMER %

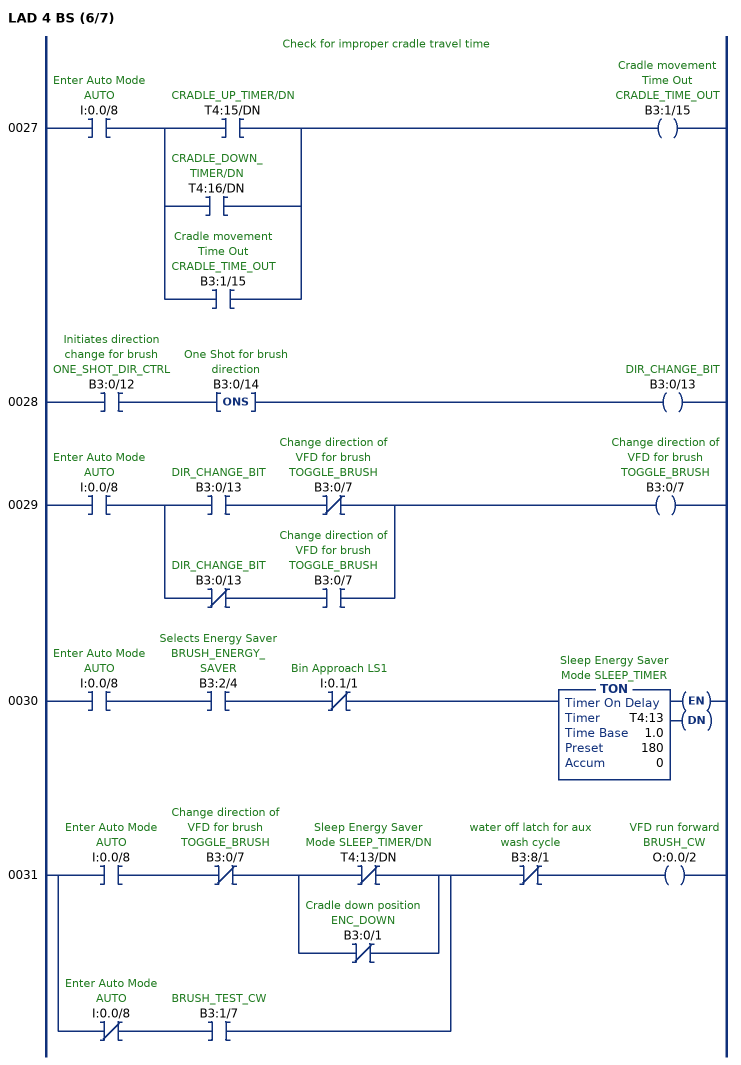
% Rung: 27 %
% Check for improper cradle travel time %
SOR XIC I:0.0/8 BST BST XIC T4:15/DN NXB XIC T4:16/DN BND NXB XIC B3:1/15 BND OTE B3:1/15 EOR
%   I:0.0/8  AUTO  "Enter Auto Mode" %
%   T4:15  CRADLE_UP_TIMER %
%   T4:16  CRADLE_DOWN_TIMER %
%   B3:1/15  CRADLE_TIME_OUT  "Cradle movement Time Out" %
% Rung: 28 %
SOR XIC B3:0/12 ONS B3:0/14 OTE B3:0/13 EOR
%   B3:0/12  ONE_SHOT_DIR_CTRL  "Initiates direction change for brush" %
%   B3:0/14  "One Shot for brush direction" %
%   B3:0/13  DIR_CHANGE_BIT %
% Rung: 29 %
SOR XIC I:0.0/8 BST XIC B3:0/13 XIO B3:0/7 NXB XIO B3:0/13 XIC B3:0/7 BND OTE B3:0/7 EOR
%   I:0.0/8  AUTO  "Enter Auto Mode" %
%   B3:0/13  DIR_CHANGE_BIT %
%   B3:0/7  TOGGLE_BRUSH  "Change direction of VFD for brush" %
% Rung: 30 %
SOR XIC I:0.0/8 XIC B3:2/4 XIO I:0.1/1 TON T4:13 1.0 180 0 EOR
%   I:0.0/8  AUTO  "Enter Auto Mode" %
%   B3:2/4  BRUSH_ENERGY_SAVER  "Selects Energy Saver" %
%   I:0.1/1  LS1  "Bin Approach" %
%   T4:13  SLEEP_TIMER  "Sleep Energy Saver Mode" %
% Rung: 31 %
SOR BST XIC I:0.0/8 XIO B3:0/7 BST XIO T4:13/DN NXB XIO B3:0/1 BND NXB XIO I:0.0/8 XIC B3:1/7 BND XIO B3:8/1 OTE O:0.0/2 EOR
%   I:0.0/8  AUTO  "Enter Auto Mode" %
%   B3:0/7  TOGGLE_BRUSH  "Change direction of VFD for brush" %
%   T4:13  SLEEP_TIMER  "Sleep Energy Saver Mode" %
%   B3:0/1  ENC_DOWN  "Cradle down position" %
%   B3:1/7  BRUSH_TEST_CW %
%   B3:8/1  "water off latch for aux wash cycle" %
%   O:0.0/2  BRUSH_CW  "VFD run forward" %

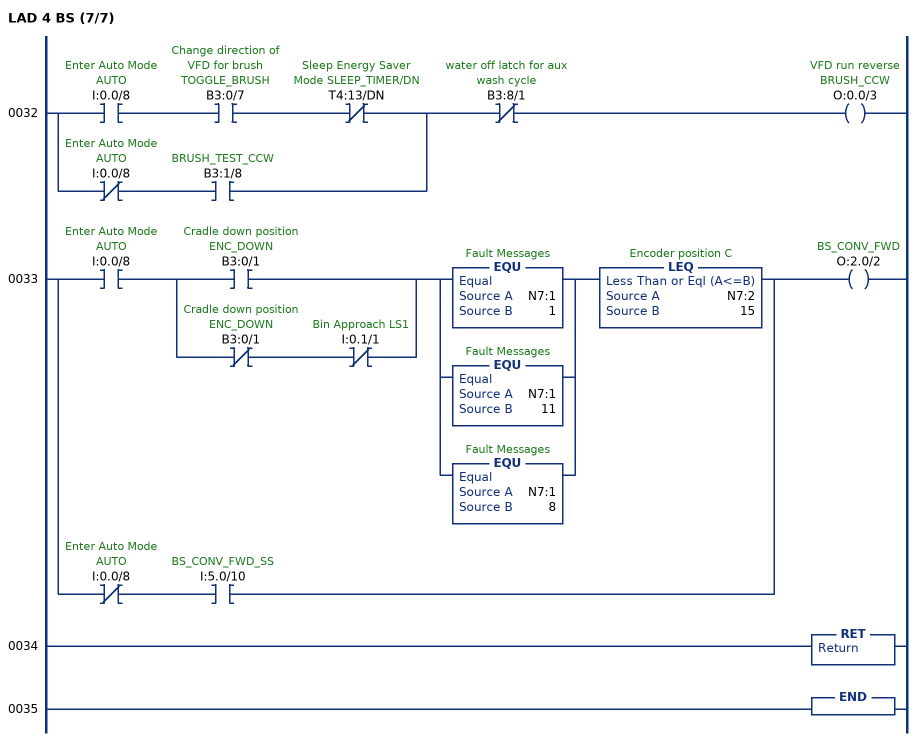
% Rung: 32 %
SOR BST XIC I:0.0/8 XIC B3:0/7 XIO T4:13/DN NXB XIO I:0.0/8 XIC B3:1/8 BND XIO B3:8/1 OTE O:0.0/3 EOR
%   I:0.0/8  AUTO  "Enter Auto Mode" %
%   B3:0/7  TOGGLE_BRUSH  "Change direction of VFD for brush" %
%   T4:13  SLEEP_TIMER  "Sleep Energy Saver Mode" %
%   B3:1/8  BRUSH_TEST_CCW %
%   B3:8/1  "water off latch for aux wash cycle" %
%   O:0.0/3  BRUSH_CCW  "VFD run reverse" %
% Rung: 33 %
SOR BST XIC I:0.0/8 BST XIC B3:0/1 NXB XIO B3:0/1 XIO I:0.1/1 BND BST EQU N7:1 1 NXB BST EQU N7:1 11 NXB EQU N7:1 8 BND BND LEQ N7:2 15 NXB XIO I:0.0/8 XIC I:5.0/10 BND OTE O:2.0/2 EOR
%   I:0.0/8  AUTO  "Enter Auto Mode" %
%   B3:0/1  ENC_DOWN  "Cradle down position" %
%   I:0.1/1  LS1  "Bin Approach" %
%   N7:1  "Fault Messages" %
%   N7:2  C  "Encoder position" %
%   I:5.0/10  BS_CONV_FWD_SS %
%   O:2.0/2  BS_CONV_FWD %
% Rung: 34 %
SOR RET EOR
% Rung: 35 %
SOR END EOR

LADDER 5 "STACKER"
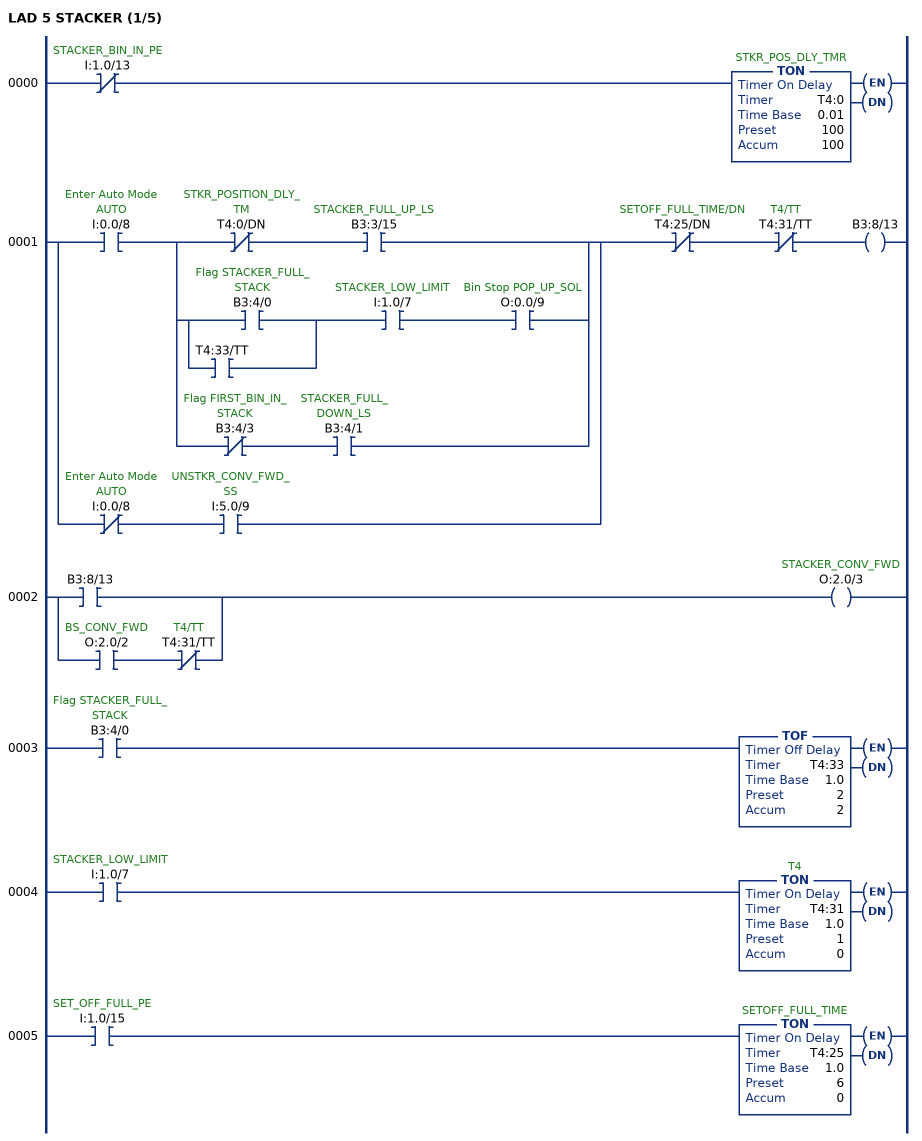
% Rung: 0 %
SOR XIO I:1.0/13 TON T4:0 0.01 100 100 EOR
%   I:1.0/13  STACKER_BIN_IN_PE %
%   T4:0  STKR_POS_DLY_TMR %
% Rung: 1 %
SOR BST XIC I:0.0/8 BST XIO T4:0/DN XIC B3:3/15 NXB BST BST XIC B3:4/0 NXB XIC T4:33/TT BND XIC I:1.0/7 XIC O:0.0/9 NXB XIO B3:4/3 XIC B3:4/1 BND BND NXB XIO I:0.0/8 XIC I:5.0/9 BND XIO T4:25/DN XIO T4:31/TT OTE B3:8/13 EOR
%   I:0.0/8  AUTO  "Enter Auto Mode" %
%   T4:0/DN  STKR_POSITION_DLY_TM %
%   B3:3/15  STACKER_FULL_UP_LS %
%   B3:4/0  STACKER_FULL_STACK  "Flag" %
%   I:1.0/7  STACKER_LOW_LIMIT %
%   O:0.0/9  POP_UP_SOL  "Bin Stop" %
%   B3:4/3  FIRST_BIN_IN_STACK  "Flag" %
%   B3:4/1  STACKER_FULL_DOWN_LS %
%   I:5.0/9  UNSTKR_CONV_FWD_SS %
%   T4:25  SETOFF_FULL_TIME %
%   T4:31  T4 %
% Rung: 2 %
SOR BST XIC B3:8/13 NXB XIC O:2.0/2 XIO T4:31/TT BND OTE O:2.0/3 EOR
%   O:2.0/2  BS_CONV_FWD %
%   T4:31  T4 %
%   O:2.0/3  STACKER_CONV_FWD %
% Rung: 3 %
SOR XIC B3:4/0 TOF T4:33 1.0 2 2 EOR
%   B3:4/0  STACKER_FULL_STACK  "Flag" %
% Rung: 4 %
SOR XIC I:1.0/7 TON T4:31 1.0 1 0 EOR
%   I:1.0/7  STACKER_LOW_LIMIT %
%   T4:31  T4 %
% Rung: 5 %
SOR XIC I:1.0/15 TON T4:25 1.0 6 0 EOR
%   I:1.0/15  SET_OFF_FULL_PE %
%   T4:25  SETOFF_FULL_TIME %

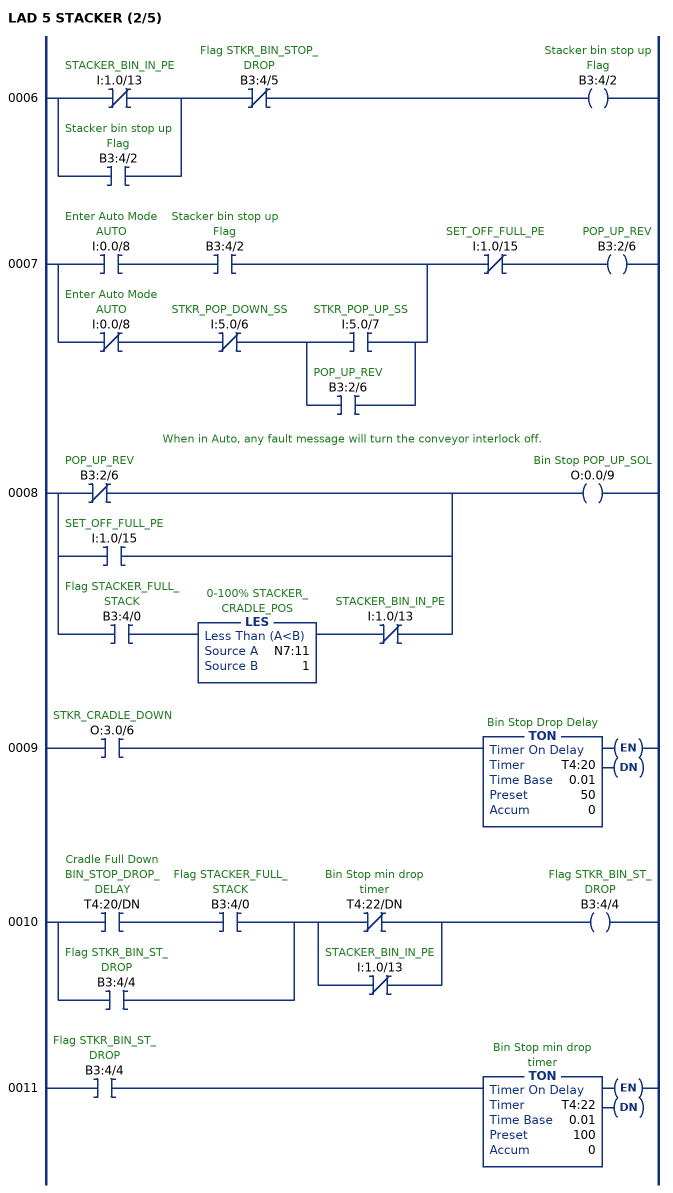
% Rung: 6 %
SOR BST XIO I:1.0/13 NXB XIC B3:4/2 BND XIO B3:4/5 OTE B3:4/2 EOR
%   I:1.0/13  STACKER_BIN_IN_PE %
%   B3:4/2  "Stacker bin stop up Flag" %
%   B3:4/5  STKR_BIN_STOP_DROP  "Flag" %
% Rung: 7 %
SOR BST XIC I:0.0/8 XIC B3:4/2 NXB XIO I:0.0/8 XIO I:5.0/6 BST XIC I:5.0/7 NXB XIC B3:2/6 BND BND XIO I:1.0/15 OTE B3:2/6 EOR
%   I:0.0/8  AUTO  "Enter Auto Mode" %
%   B3:4/2  "Stacker bin stop up Flag" %
%   I:5.0/6  STKR_POP_DOWN_SS %
%   I:5.0/7  STKR_POP_UP_SS %
%   B3:2/6  POP_UP_REV %
%   I:1.0/15  SET_OFF_FULL_PE %
% Rung: 8 %
% When in Auto, any fault message will turn the conveyor interlock off. %
SOR BST XIO B3:2/6 NXB BST XIC I:1.0/15 NXB XIC B3:4/0 LES N7:11 1 XIO I:1.0/13 BND BND OTE O:0.0/9 EOR
%   B3:2/6  POP_UP_REV %
%   I:1.0/15  SET_OFF_FULL_PE %
%   B3:4/0  STACKER_FULL_STACK  "Flag" %
%   N7:11  STACKER_CRADLE_POS  "0-100%" %
%   I:1.0/13  STACKER_BIN_IN_PE %
%   O:0.0/9  POP_UP_SOL  "Bin Stop" %
% Rung: 9 %
SOR XIC O:3.0/6 TON T4:20 0.01 50 0 EOR
%   O:3.0/6  STKR_CRADLE_DOWN %
%   T4:20  "Bin Stop Drop Delay" %
% Rung: 10 %
SOR BST XIC T4:20/DN XIC B3:4/0 NXB XIC B3:4/4 BND BST XIO T4:22/DN NXB XIO I:1.0/13 BND OTE B3:4/4 EOR
%   T4:20/DN  BIN_STOP_DROP_DELAY  "Cradle Full Down" %
%   B3:4/0  STACKER_FULL_STACK  "Flag" %
%   B3:4/4  STKR_BIN_ST_DROP  "Flag" %
%   T4:22  "Bin Stop min drop timer" %
%   I:1.0/13  STACKER_BIN_IN_PE %
% Rung: 11 %
SOR XIC B3:4/4 TON T4:22 0.01 100 0 EOR
%   B3:4/4  STKR_BIN_ST_DROP  "Flag" %
%   T4:22  "Bin Stop min drop timer" %

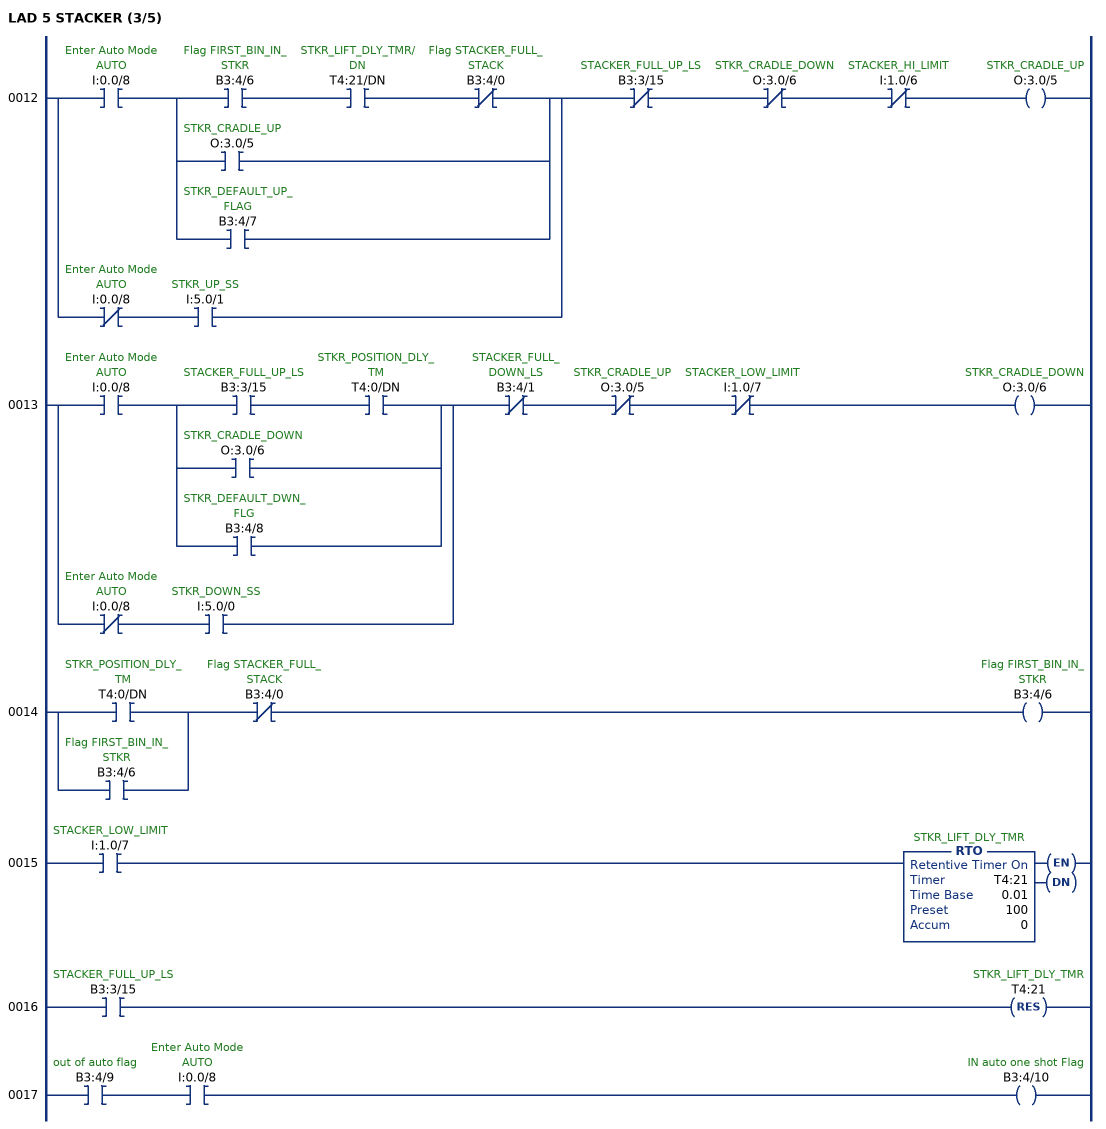
% Rung: 12 %
SOR BST XIC I:0.0/8 BST XIC B3:4/6 XIC T4:21/DN XIO B3:4/0 NXB BST XIC O:3.0/5 NXB XIC B3:4/7 BND BND NXB XIO I:0.0/8 XIC I:5.0/1 BND XIO B3:3/15 XIO O:3.0/6 XIO I:1.0/6 OTE O:3.0/5 EOR
%   I:0.0/8  AUTO  "Enter Auto Mode" %
%   B3:4/6  FIRST_BIN_IN_STKR  "Flag" %
%   T4:21  STKR_LIFT_DLY_TMR %
%   B3:4/0  STACKER_FULL_STACK  "Flag" %
%   O:3.0/5  STKR_CRADLE_UP %
%   B3:4/7  STKR_DEFAULT_UP_FLAG %
%   I:5.0/1  STKR_UP_SS %
%   B3:3/15  STACKER_FULL_UP_LS %
%   O:3.0/6  STKR_CRADLE_DOWN %
%   I:1.0/6  STACKER_HI_LIMIT %
% Rung: 13 %
SOR BST XIC I:0.0/8 BST XIC B3:3/15 XIC T4:0/DN NXB BST XIC O:3.0/6 NXB XIC B3:4/8 BND BND NXB XIO I:0.0/8 XIC I:5.0/0 BND XIO B3:4/1 XIO O:3.0/5 XIO I:1.0/7 OTE O:3.0/6 EOR
%   I:0.0/8  AUTO  "Enter Auto Mode" %
%   B3:3/15  STACKER_FULL_UP_LS %
%   T4:0/DN  STKR_POSITION_DLY_TM %
%   O:3.0/6  STKR_CRADLE_DOWN %
%   B3:4/8  STKR_DEFAULT_DWN_FLG %
%   I:5.0/0  STKR_DOWN_SS %
%   B3:4/1  STACKER_FULL_DOWN_LS %
%   O:3.0/5  STKR_CRADLE_UP %
%   I:1.0/7  STACKER_LOW_LIMIT %
% Rung: 14 %
SOR BST XIC T4:0/DN NXB XIC B3:4/6 BND XIO B3:4/0 OTE B3:4/6 EOR
%   T4:0/DN  STKR_POSITION_DLY_TM %
%   B3:4/6  FIRST_BIN_IN_STKR  "Flag" %
%   B3:4/0  STACKER_FULL_STACK  "Flag" %
% Rung: 15 %
SOR XIC I:1.0/7 RTO T4:21 0.01 100 0 EOR
%   I:1.0/7  STACKER_LOW_LIMIT %
%   T4:21  STKR_LIFT_DLY_TMR %
% Rung: 16 %
SOR XIC B3:3/15 RES T4:21 EOR
%   B3:3/15  STACKER_FULL_UP_LS %
%   T4:21  STKR_LIFT_DLY_TMR %
% Rung: 17 %
SOR XIC B3:4/9 XIC I:0.0/8 OTE B3:4/10 EOR
%   B3:4/9  "out of auto flag" %
%   I:0.0/8  AUTO  "Enter Auto Mode" %
%   B3:4/10  "IN auto one shot Flag" %

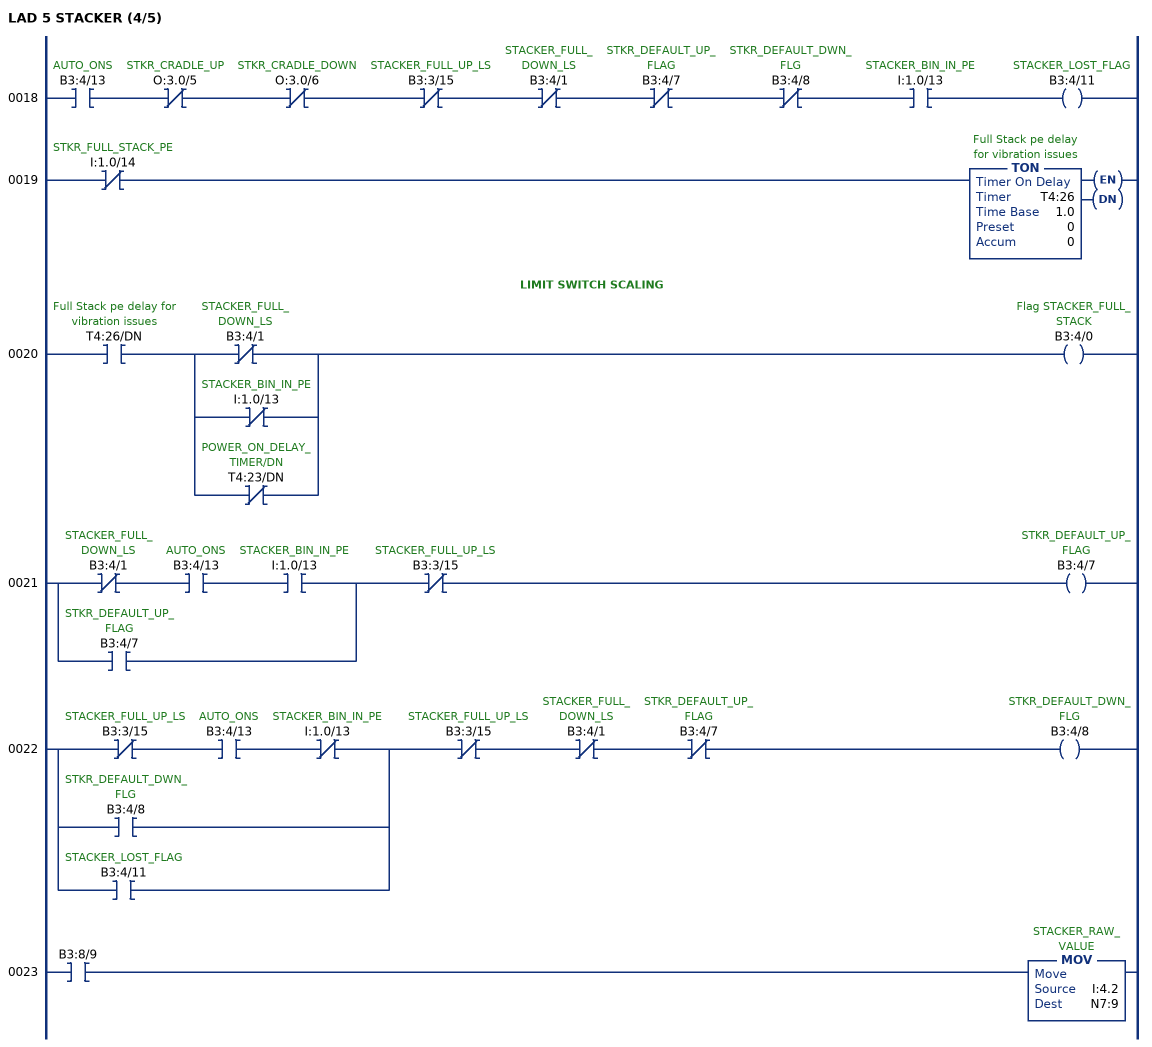
% Rung: 18 %
SOR XIC B3:4/13 XIO O:3.0/5 XIO O:3.0/6 XIO B3:3/15 XIO B3:4/1 XIO B3:4/7 XIO B3:4/8 XIC I:1.0/13 OTE B3:4/11 EOR
%   B3:4/13  AUTO_ONS %
%   O:3.0/5  STKR_CRADLE_UP %
%   O:3.0/6  STKR_CRADLE_DOWN %
%   B3:3/15  STACKER_FULL_UP_LS %
%   B3:4/1  STACKER_FULL_DOWN_LS %
%   B3:4/7  STKR_DEFAULT_UP_FLAG %
%   B3:4/8  STKR_DEFAULT_DWN_FLG %
%   I:1.0/13  STACKER_BIN_IN_PE %
%   B3:4/11  STACKER_LOST_FLAG %
% Rung: 19 %
SOR XIO I:1.0/14 TON T4:26 1.0 0 0 EOR
%   I:1.0/14  STKR_FULL_STACK_PE %
%   T4:26  "Full Stack pe delay for vibration issues" %
% Rung: 20 %
% TITLE: LIMIT SWITCH SCALING %
SOR XIC T4:26/DN BST XIO B3:4/1 NXB BST XIO I:1.0/13 NXB XIO T4:23/DN BND BND OTE B3:4/0 EOR
%   T4:26  "Full Stack pe delay for vibration issues" %
%   B3:4/1  STACKER_FULL_DOWN_LS %
%   I:1.0/13  STACKER_BIN_IN_PE %
%   T4:23  POWER_ON_DELAY_TIMER %
%   B3:4/0  STACKER_FULL_STACK  "Flag" %
% Rung: 21 %
SOR BST XIO B3:4/1 XIC B3:4/13 XIC I:1.0/13 NXB XIC B3:4/7 BND XIO B3:3/15 OTE B3:4/7 EOR
%   B3:4/1  STACKER_FULL_DOWN_LS %
%   B3:4/13  AUTO_ONS %
%   I:1.0/13  STACKER_BIN_IN_PE %
%   B3:4/7  STKR_DEFAULT_UP_FLAG %
%   B3:3/15  STACKER_FULL_UP_LS %
% Rung: 22 %
SOR BST XIO B3:3/15 XIC B3:4/13 XIO I:1.0/13 NXB BST XIC B3:4/8 NXB XIC B3:4/11 BND BND XIO B3:3/15 XIO B3:4/1 XIO B3:4/7 OTE B3:4/8 EOR
%   B3:3/15  STACKER_FULL_UP_LS %
%   B3:4/13  AUTO_ONS %
%   I:1.0/13  STACKER_BIN_IN_PE %
%   B3:4/8  STKR_DEFAULT_DWN_FLG %
%   B3:4/11  STACKER_LOST_FLAG %
%   B3:4/1  STACKER_FULL_DOWN_LS %
%   B3:4/7  STKR_DEFAULT_UP_FLAG %
% Rung: 23 %
SOR XIC B3:8/9 MOV I:4.2 N7:9 EOR
%   N7:9  STACKER_RAW_VALUE %

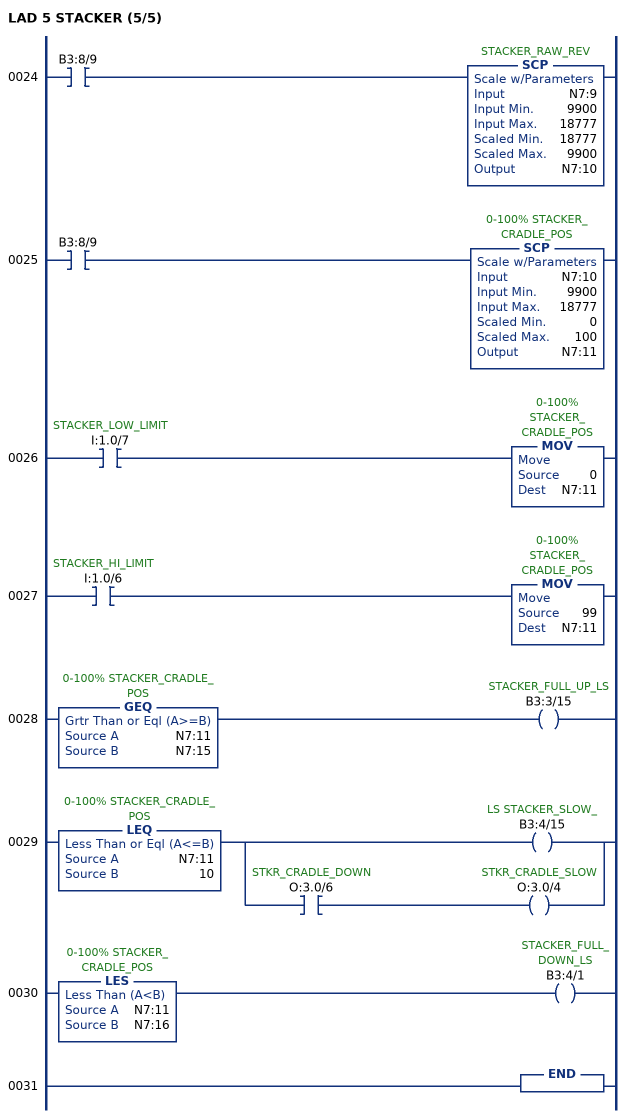
% Rung: 24 %
SOR XIC B3:8/9 SCP N7:9 9900 18777 18777 9900 N7:10 EOR
%   N7:9  STACKER_RAW_VALUE %
%   N7:10  STACKER_RAW_REV %
% Rung: 25 %
SOR XIC B3:8/9 SCP N7:10 9900 18777 0 100 N7:11 EOR
%   N7:10  STACKER_RAW_REV %
%   N7:11  STACKER_CRADLE_POS  "0-100%" %
% Rung: 26 %
SOR XIC I:1.0/7 MOV 0 N7:11 EOR
%   I:1.0/7  STACKER_LOW_LIMIT %
%   N7:11  STACKER_CRADLE_POS  "0-100%" %
% Rung: 27 %
SOR XIC I:1.0/6 MOV 99 N7:11 EOR
%   I:1.0/6  STACKER_HI_LIMIT %
%   N7:11  STACKER_CRADLE_POS  "0-100%" %
% Rung: 28 %
SOR GEQ N7:11 N7:15 OTE B3:3/15 EOR
%   N7:11  STACKER_CRADLE_POS  "0-100%" %
%   N7:15  STKR_FULL_UP_SP  "Stacker Full Up" %
%   B3:3/15  STACKER_FULL_UP_LS %
% Rung: 29 %
SOR LEQ N7:11 10 BST OTE B3:4/15 NXB XIC O:3.0/6 OTE O:3.0/4 BND EOR
%   N7:11  STACKER_CRADLE_POS  "0-100%" %
%   B3:4/15  STACKER_SLOW_  "LS" %
%   O:3.0/6  STKR_CRADLE_DOWN %
%   O:3.0/4  STKR_CRADLE_SLOW %
% Rung: 30 %
SOR LES N7:11 N7:16 OTE B3:4/1 EOR
%   N7:11  STACKER_CRADLE_POS  "0-100%" %
%   N7:16  STKR_FULL_DOWN_SP  "Stacker FUll Down" %
%   B3:4/1  STACKER_FULL_DOWN_LS %
% Rung: 31 %
SOR END EOR

LADDER 6 "WATER"
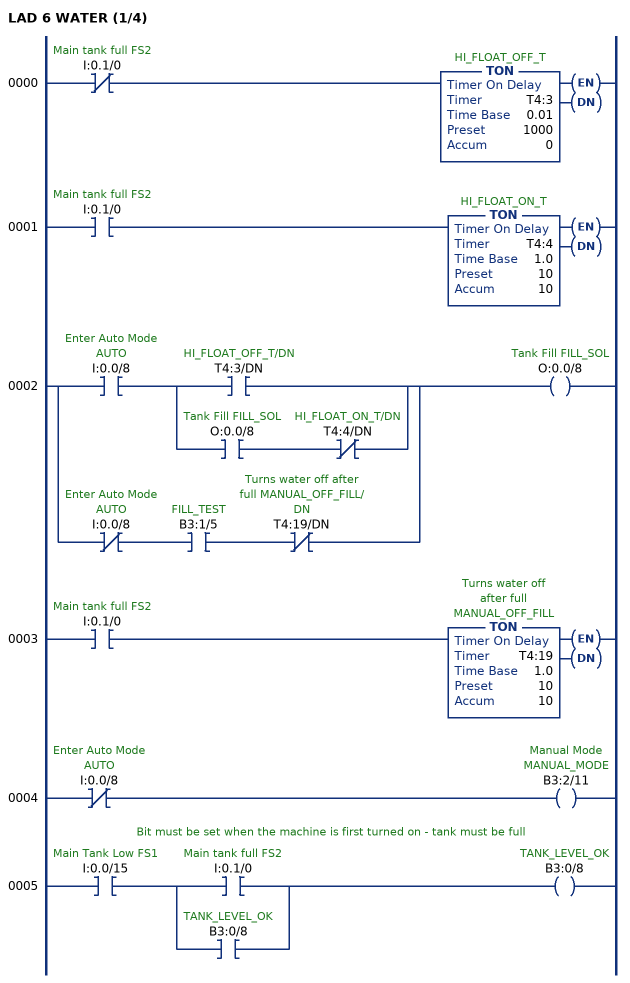
% Rung: 0 %
SOR XIO I:0.1/0 TON T4:3 0.01 1000 0 EOR
%   I:0.1/0  FS2  "Main tank full" %
%   T4:3  HI_FLOAT_OFF_T %
% Rung: 1 %
SOR XIC I:0.1/0 TON T4:4 1.0 10 10 EOR
%   I:0.1/0  FS2  "Main tank full" %
%   T4:4  HI_FLOAT_ON_T %
% Rung: 2 %
SOR BST XIC I:0.0/8 BST XIC T4:3/DN NXB XIC O:0.0/8 XIO T4:4/DN BND NXB XIO I:0.0/8 XIC B3:1/5 XIO T4:19/DN BND OTE O:0.0/8 EOR
%   I:0.0/8  AUTO  "Enter Auto Mode" %
%   T4:3  HI_FLOAT_OFF_T %
%   O:0.0/8  FILL_SOL  "Tank Fill" %
%   T4:4  HI_FLOAT_ON_T %
%   B3:1/5  FILL_TEST %
%   T4:19  MANUAL_OFF_FILL  "Turns water off after full" %
% Rung: 3 %
SOR XIC I:0.1/0 TON T4:19 1.0 10 10 EOR
%   I:0.1/0  FS2  "Main tank full" %
%   T4:19  MANUAL_OFF_FILL  "Turns water off after full" %
% Rung: 4 %
SOR XIO I:0.0/8 OTE B3:2/11 EOR
%   I:0.0/8  AUTO  "Enter Auto Mode" %
%   B3:2/11  MANUAL_MODE  "Manual Mode" %
% Rung: 5 %
% Bit must be set when the machine is first turned on - tank must be full %
SOR XIC I:0.0/15 BST XIC I:0.1/0 NXB XIC B3:0/8 BND OTE B3:0/8 EOR
%   I:0.0/15  FS1  "Main Tank Low" %
%   I:0.1/0  FS2  "Main tank full" %
%   B3:0/8  TANK_LEVEL_OK %

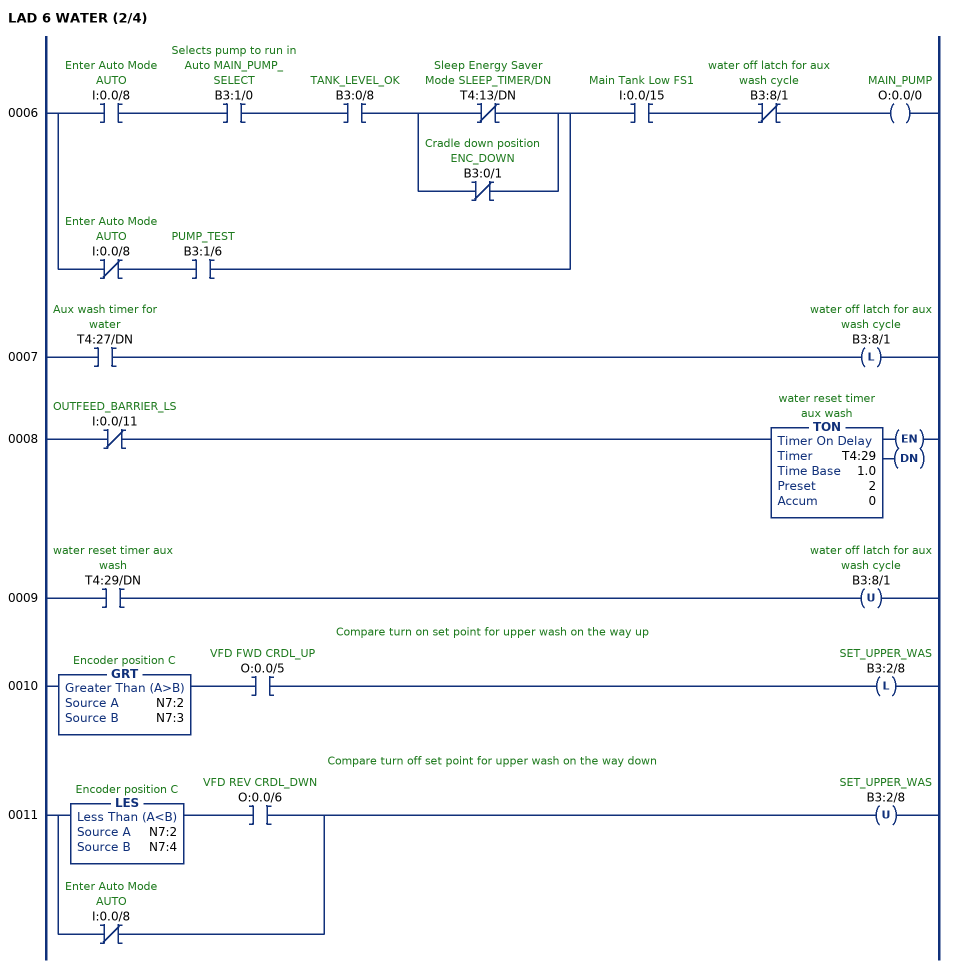
% Rung: 6 %
SOR BST XIC I:0.0/8 XIC B3:1/0 XIC B3:0/8 BST XIO T4:13/DN NXB XIO B3:0/1 BND NXB XIO I:0.0/8 XIC B3:1/6 BND XIC I:0.0/15 XIO B3:8/1 OTE O:0.0/0 EOR
%   I:0.0/8  AUTO  "Enter Auto Mode" %
%   B3:1/0  MAIN_PUMP_SELECT  "Selects pump to run in Auto" %
%   B3:0/8  TANK_LEVEL_OK %
%   T4:13  SLEEP_TIMER  "Sleep Energy Saver Mode" %
%   B3:0/1  ENC_DOWN  "Cradle down position" %
%   B3:1/6  PUMP_TEST %
%   I:0.0/15  FS1  "Main Tank Low" %
%   B3:8/1  "water off latch for aux wash cycle" %
%   O:0.0/0  MAIN_PUMP %
% Rung: 7 %
SOR XIC T4:27/DN OTL B3:8/1 EOR
%   T4:27  "Aux wash timer for water" %
%   B3:8/1  "water off latch for aux wash cycle" %
% Rung: 8 %
SOR XIO I:0.0/11 TON T4:29 1.0 2 0 EOR
%   I:0.0/11  OUTFEED_BARRIER_LS %
%   T4:29  "water reset timer aux wash" %
% Rung: 9 %
SOR XIC T4:29/DN OTU B3:8/1 EOR
%   T4:29  "water reset timer aux wash" %
%   B3:8/1  "water off latch for aux wash cycle" %
% Rung: 10 %
% Compare turn on set point for upper wash on the way up %
SOR GRT N7:2 N7:3 XIC O:0.0/5 OTL B3:2/8 EOR
%   N7:2  C  "Encoder position" %
%   N7:3  UPPER_WASH_TURN_ON %
%   O:0.0/5  CRDL_UP  "VFD FWD" %
%   B3:2/8  SET_UPPER_WAS %
% Rung: 11 %
% Compare turn off set point for upper wash on the way down %
SOR BST LES N7:2 N7:4 XIC O:0.0/6 NXB XIO I:0.0/8 BND OTU B3:2/8 EOR
%   N7:2  C  "Encoder position" %
%   N7:4  UPPER_WASH_TURN_OFF %
%   O:0.0/6  CRDL_DWN  "VFD REV" %
%   I:0.0/8  AUTO  "Enter Auto Mode" %
%   B3:2/8  SET_UPPER_WAS %

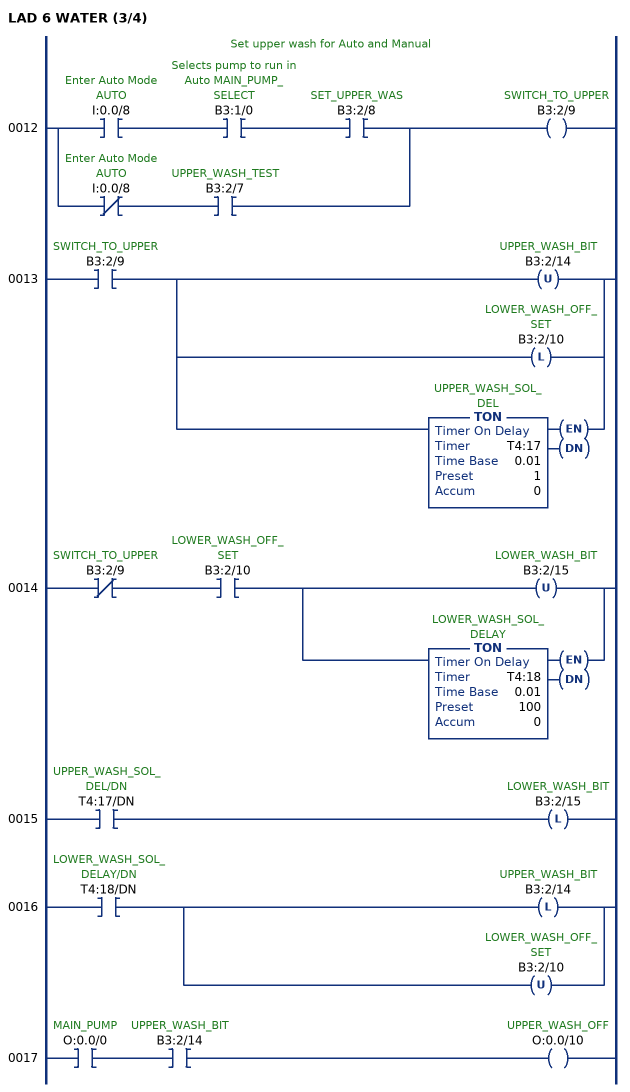
% Rung: 12 %
% Set upper wash for Auto and Manual %
SOR BST XIC I:0.0/8 XIC B3:1/0 XIC B3:2/8 NXB XIO I:0.0/8 XIC B3:2/7 BND OTE B3:2/9 EOR
%   I:0.0/8  AUTO  "Enter Auto Mode" %
%   B3:1/0  MAIN_PUMP_SELECT  "Selects pump to run in Auto" %
%   B3:2/8  SET_UPPER_WAS %
%   B3:2/7  UPPER_WASH_TEST %
%   B3:2/9  SWITCH_TO_UPPER %
% Rung: 13 %
SOR XIC B3:2/9 BST OTU B3:2/14 NXB BST OTL B3:2/10 NXB TON T4:17 0.01 1 0 BND BND EOR
%   B3:2/9  SWITCH_TO_UPPER %
%   B3:2/14  UPPER_WASH_BIT %
%   B3:2/10  LOWER_WASH_OFF_SET %
%   T4:17  UPPER_WASH_SOL_DEL %
% Rung: 14 %
SOR XIO B3:2/9 XIC B3:2/10 BST OTU B3:2/15 NXB TON T4:18 0.01 100 0 BND EOR
%   B3:2/9  SWITCH_TO_UPPER %
%   B3:2/10  LOWER_WASH_OFF_SET %
%   B3:2/15  LOWER_WASH_BIT %
%   T4:18  LOWER_WASH_SOL_DELAY %
% Rung: 15 %
SOR XIC T4:17/DN OTL B3:2/15 EOR
%   T4:17  UPPER_WASH_SOL_DEL %
%   B3:2/15  LOWER_WASH_BIT %
% Rung: 16 %
SOR XIC T4:18/DN BST OTL B3:2/14 NXB OTU B3:2/10 BND EOR
%   T4:18  LOWER_WASH_SOL_DELAY %
%   B3:2/14  UPPER_WASH_BIT %
%   B3:2/10  LOWER_WASH_OFF_SET %
% Rung: 17 %
SOR XIC O:0.0/0 XIC B3:2/14 OTE O:0.0/10 EOR
%   O:0.0/0  MAIN_PUMP %
%   B3:2/14  UPPER_WASH_BIT %
%   O:0.0/10  UPPER_WASH_OFF %

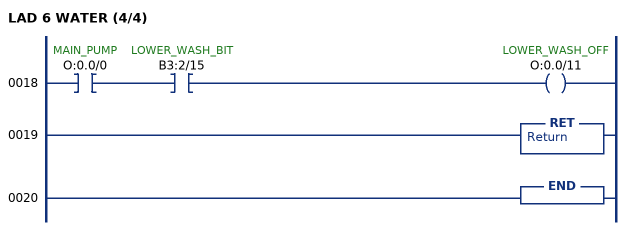
% Rung: 18 %
SOR XIC O:0.0/0 XIC B3:2/15 OTE O:0.0/11 EOR
%   O:0.0/0  MAIN_PUMP %
%   B3:2/15  LOWER_WASH_BIT %
%   O:0.0/11  LOWER_WASH_OFF %
% Rung: 19 %
SOR RET EOR
% Rung: 20 %
SOR END EOR

LADDER 8 "ENCODER"    % Bin Scrubber HSC %
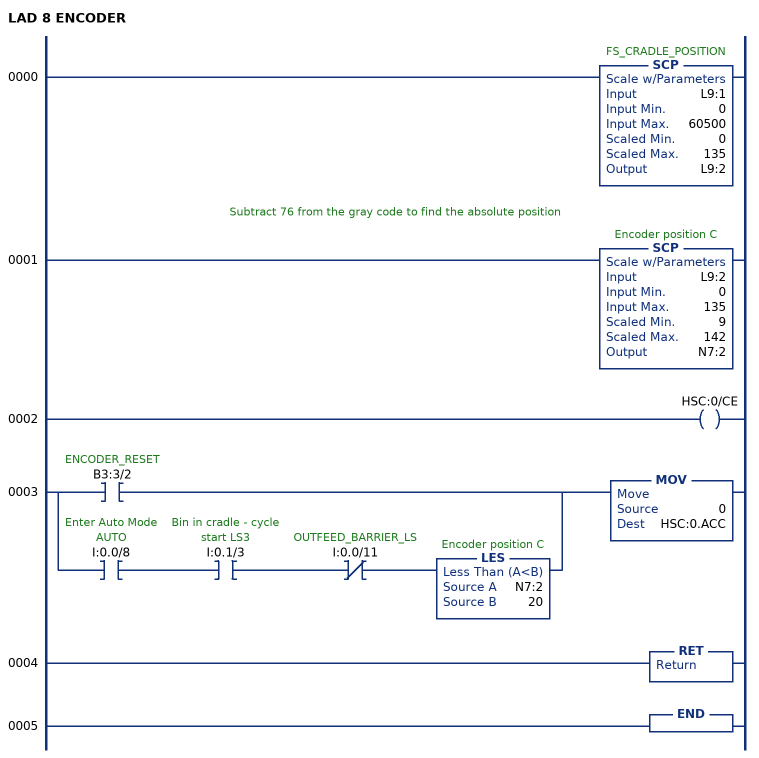
% Rung: 0 %
SOR SCP L9:1 0 60500 0 135 L9:2 EOR
%   L9:1  HSC_RAW_ACC %
%   L9:2  FS_CRADLE_POSITION %
% Rung: 1 %
% Subtract 76 from the gray code to find the absolute position %
SOR SCP L9:2 0 135 9 142 N7:2 EOR
%   L9:2  FS_CRADLE_POSITION %
%   N7:2  C  "Encoder position" %
% Rung: 2 %
SOR OTE HSC:0/CE EOR
% Rung: 3 %
SOR BST XIC B3:3/2 NXB XIC I:0.0/8 XIC I:0.1/3 XIO I:0.0/11 LES N7:2 20 BND MOV 0 HSC:0.ACC EOR
%   B3:3/2  ENCODER_RESET %
%   I:0.0/8  AUTO  "Enter Auto Mode" %
%   I:0.1/3  LS3  "Bin in cradle - cycle start" %
%   I:0.0/11  OUTFEED_BARRIER_LS %
%   N7:2  C  "Encoder position" %
% Rung: 4 %
SOR RET EOR
% Rung: 5 %
SOR END EOR

LADDER 9 "STARTUP"
